// TIA Portal V17 export
// export: Created 2023-04-26T11:43:36.2466218Z, ExportSetting None, DisplayName Totally Integrated Automation Portal, DisplayVersion V17 Update 4, DisplayName TIA Portal Openness, DisplayVersion V17 Update 4, DisplayName TIA Portal Version Control Interface, DisplayVersion V17, DisplayName STEP 7 Professional, DisplayVersion V17 Update 4, DisplayName STEP 7 Safety, DisplayVersion V17, DisplayName WinCC Advanced / Unified PC, DisplayVersion V17 Update 4
FUNCTION "FC_AIn" : Void   // FC14, LAD
TITLE = FC_AIn
{ S7_Optimized_Access := 'FALSE' }
// Analog Input
// stored: SetENOAutomatically false
BEGIN

REGION Network 1: COMPRESSOR SUCTION PRESSURE
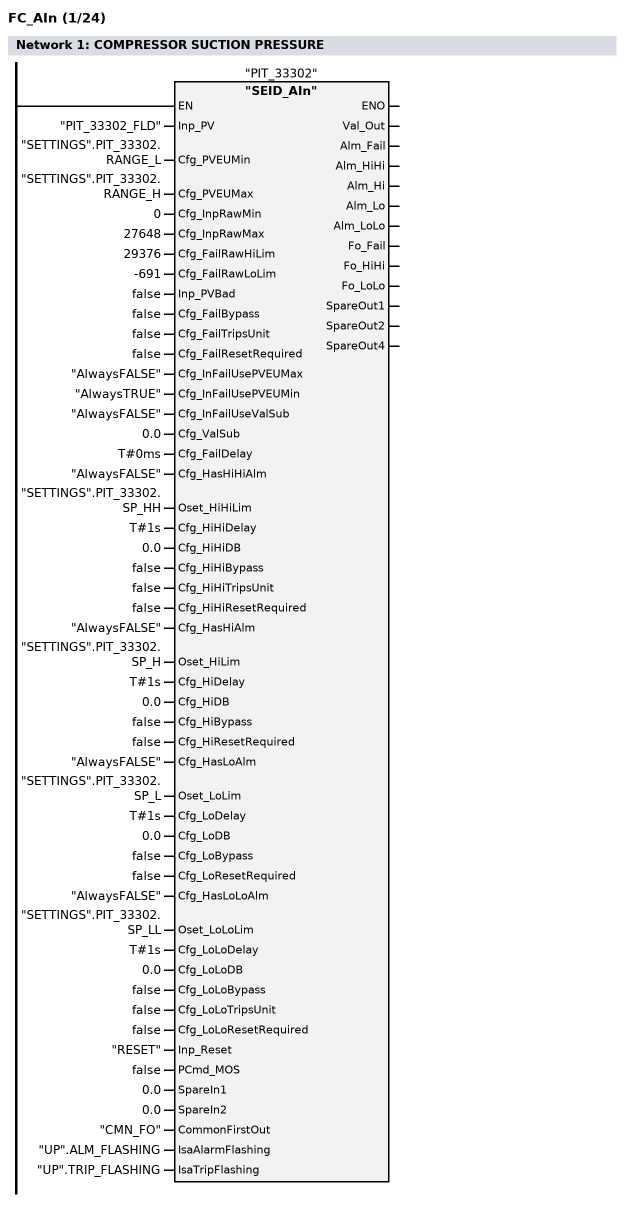
   RUNG wire#powerrail
      "PIT_33302"(Inp_PV := "PIT_33302_FLD", Cfg_PVEUMin := "SETTINGS".PIT_33302.RANGE_L, Cfg_PVEUMax := "SETTINGS".PIT_33302.RANGE_H, Cfg_InpRawMin := 0, Cfg_InpRawMax := 27648, Cfg_FailRawHiLim := 29376, Cfg_FailRawLoLim := -691, Inp_PVBad := false, Cfg_FailBypass := false, Cfg_FailTripsUnit := false, Cfg_FailResetRequired := false, Cfg_InFailUsePVEUMax := "AlwaysFALSE", Cfg_InFailUsePVEUMin := "AlwaysTRUE", Cfg_InFailUseValSub := "AlwaysFALSE", Cfg_ValSub := 0.0, Cfg_FailDelay := T#0ms, Cfg_HasHiHiAlm := "AlwaysFALSE", Oset_HiHiLim := "SETTINGS".PIT_33302.SP_HH, Cfg_HiHiDelay := T#1s, Cfg_HiHiDB := 0.0, Cfg_HiHiBypass := false, Cfg_HiHiTripsUnit := false, Cfg_HiHiResetRequired := false, Cfg_HasHiAlm := "AlwaysFALSE", Oset_HiLim := "SETTINGS".PIT_33302.SP_H, Cfg_HiDelay := T#1s, Cfg_HiDB := 0.0, Cfg_HiBypass := false, Cfg_HiResetRequired := false, Cfg_HasLoAlm := "AlwaysFALSE", Oset_LoLim := "SETTINGS".PIT_33302.SP_L, Cfg_LoDelay := T#1s, Cfg_LoDB := 0.0, Cfg_LoBypass := false, Cfg_LoResetRequired := false, Cfg_HasLoLoAlm := "AlwaysFALSE", Oset_LoLoLim := "SETTINGS".PIT_33302.SP_LL, Cfg_LoLoDelay := T#1s, Cfg_LoLoDB := 0.0, Cfg_LoLoBypass := false, Cfg_LoLoTripsUnit := false, Cfg_LoLoResetRequired := false, Inp_Reset := "RESET", PCmd_MOS := false, SpareIn1 := 0.0, SpareIn2 := 0.0, CommonFirstOut := "CMN_FO", IsaAlarmFlashing := "UP".ALM_FLASHING, IsaTripFlashing := "UP".TRIP_FLASHING, Val_Out =>, Alm_Fail =>, Alm_HiHi =>, Alm_Hi =>, Alm_Lo =>, Alm_LoLo =>, Fo_Fail =>, Fo_HiHi =>, Fo_LoLo =>, SpareOut1 =>, SpareOut2 =>, SpareOut4 =>)
   END_RUNG
   // the same network as SCL:
   "PIT_33302"(Inp_PV := "PIT_33302_FLD",   // "SEID_AIn"
               Cfg_PVEUMin := "SETTINGS".PIT_33302.RANGE_L,
               Cfg_PVEUMax := "SETTINGS".PIT_33302.RANGE_H,
               Cfg_InpRawMin := 0,
               Cfg_InpRawMax := 27648,
               Cfg_FailRawHiLim := 29376,
               Cfg_FailRawLoLim := -691,
               Inp_PVBad := false,
               Cfg_FailBypass := false,
               Cfg_FailTripsUnit := false,
               Cfg_FailResetRequired := false,
               Cfg_InFailUsePVEUMax := "AlwaysFALSE",
               Cfg_InFailUsePVEUMin := "AlwaysTRUE",
               Cfg_InFailUseValSub := "AlwaysFALSE",
               Cfg_ValSub := 0.0,
               Cfg_FailDelay := T#0ms,
               Cfg_HasHiHiAlm := "AlwaysFALSE",
               Oset_HiHiLim := "SETTINGS".PIT_33302.SP_HH,
               Cfg_HiHiDelay := T#1s,
               Cfg_HiHiDB := 0.0,
               Cfg_HiHiBypass := false,
               Cfg_HiHiTripsUnit := false,
               Cfg_HiHiResetRequired := false,
               Cfg_HasHiAlm := "AlwaysFALSE",
               Oset_HiLim := "SETTINGS".PIT_33302.SP_H,
               Cfg_HiDelay := T#1s,
               Cfg_HiDB := 0.0,
               Cfg_HiBypass := false,
               Cfg_HiResetRequired := false,
               Cfg_HasLoAlm := "AlwaysFALSE",
               Oset_LoLim := "SETTINGS".PIT_33302.SP_L,
               Cfg_LoDelay := T#1s,
               Cfg_LoDB := 0.0,
               Cfg_LoBypass := false,
               Cfg_LoResetRequired := false,
               Cfg_HasLoLoAlm := "AlwaysFALSE",
               Oset_LoLoLim := "SETTINGS".PIT_33302.SP_LL,
               Cfg_LoLoDelay := T#1s,
               Cfg_LoLoDB := 0.0,
               Cfg_LoLoBypass := false,
               Cfg_LoLoTripsUnit := false,
               Cfg_LoLoResetRequired := false,
               Inp_Reset := "RESET",
               PCmd_MOS := false,
               SpareIn1 := 0.0,
               SpareIn2 := 0.0,
               CommonFirstOut := "CMN_FO",
               IsaAlarmFlashing := "UP".ALM_FLASHING,
               IsaTripFlashing := "UP".TRIP_FLASHING);
END_REGION

REGION Network 2: LUBE OIL SEPARATOR OUTLET PRESSURE
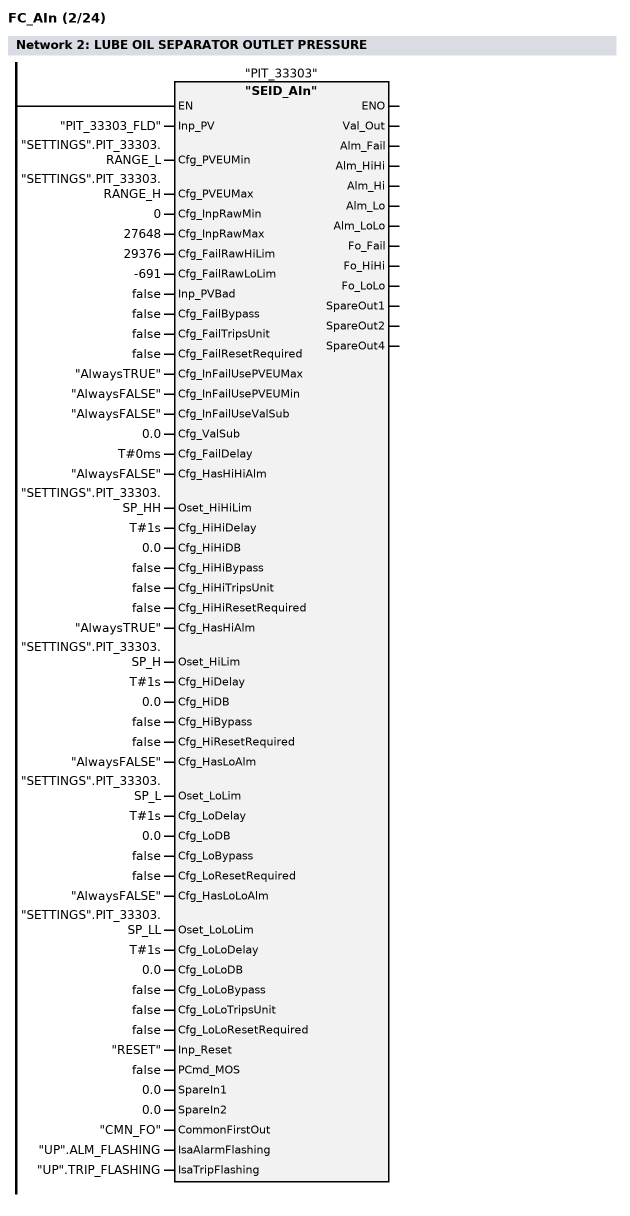
   RUNG wire#powerrail
      "PIT_33303"(Inp_PV := "PIT_33303_FLD", Cfg_PVEUMin := "SETTINGS".PIT_33303.RANGE_L, Cfg_PVEUMax := "SETTINGS".PIT_33303.RANGE_H, Cfg_InpRawMin := 0, Cfg_InpRawMax := 27648, Cfg_FailRawHiLim := 29376, Cfg_FailRawLoLim := -691, Inp_PVBad := false, Cfg_FailBypass := false, Cfg_FailTripsUnit := false, Cfg_FailResetRequired := false, Cfg_InFailUsePVEUMax := "AlwaysTRUE", Cfg_InFailUsePVEUMin := "AlwaysFALSE", Cfg_InFailUseValSub := "AlwaysFALSE", Cfg_ValSub := 0.0, Cfg_FailDelay := T#0ms, Cfg_HasHiHiAlm := "AlwaysFALSE", Oset_HiHiLim := "SETTINGS".PIT_33303.SP_HH, Cfg_HiHiDelay := T#1s, Cfg_HiHiDB := 0.0, Cfg_HiHiBypass := false, Cfg_HiHiTripsUnit := false, Cfg_HiHiResetRequired := false, Cfg_HasHiAlm := "AlwaysTRUE", Oset_HiLim := "SETTINGS".PIT_33303.SP_H, Cfg_HiDelay := T#1s, Cfg_HiDB := 0.0, Cfg_HiBypass := false, Cfg_HiResetRequired := false, Cfg_HasLoAlm := "AlwaysFALSE", Oset_LoLim := "SETTINGS".PIT_33303.SP_L, Cfg_LoDelay := T#1s, Cfg_LoDB := 0.0, Cfg_LoBypass := false, Cfg_LoResetRequired := false, Cfg_HasLoLoAlm := "AlwaysFALSE", Oset_LoLoLim := "SETTINGS".PIT_33303.SP_LL, Cfg_LoLoDelay := T#1s, Cfg_LoLoDB := 0.0, Cfg_LoLoBypass := false, Cfg_LoLoTripsUnit := false, Cfg_LoLoResetRequired := false, Inp_Reset := "RESET", PCmd_MOS := false, SpareIn1 := 0.0, SpareIn2 := 0.0, CommonFirstOut := "CMN_FO", IsaAlarmFlashing := "UP".ALM_FLASHING, IsaTripFlashing := "UP".TRIP_FLASHING, Val_Out =>, Alm_Fail =>, Alm_HiHi =>, Alm_Hi =>, Alm_Lo =>, Alm_LoLo =>, Fo_Fail =>, Fo_HiHi =>, Fo_LoLo =>, SpareOut1 =>, SpareOut2 =>, SpareOut4 =>)
   END_RUNG
   // the same network as SCL:
   "PIT_33303"(Inp_PV := "PIT_33303_FLD",   // "SEID_AIn"
               Cfg_PVEUMin := "SETTINGS".PIT_33303.RANGE_L,
               Cfg_PVEUMax := "SETTINGS".PIT_33303.RANGE_H,
               Cfg_InpRawMin := 0,
               Cfg_InpRawMax := 27648,
               Cfg_FailRawHiLim := 29376,
               Cfg_FailRawLoLim := -691,
               Inp_PVBad := false,
               Cfg_FailBypass := false,
               Cfg_FailTripsUnit := false,
               Cfg_FailResetRequired := false,
               Cfg_InFailUsePVEUMax := "AlwaysTRUE",
               Cfg_InFailUsePVEUMin := "AlwaysFALSE",
               Cfg_InFailUseValSub := "AlwaysFALSE",
               Cfg_ValSub := 0.0,
               Cfg_FailDelay := T#0ms,
               Cfg_HasHiHiAlm := "AlwaysFALSE",
               Oset_HiHiLim := "SETTINGS".PIT_33303.SP_HH,
               Cfg_HiHiDelay := T#1s,
               Cfg_HiHiDB := 0.0,
               Cfg_HiHiBypass := false,
               Cfg_HiHiTripsUnit := false,
               Cfg_HiHiResetRequired := false,
               Cfg_HasHiAlm := "AlwaysTRUE",
               Oset_HiLim := "SETTINGS".PIT_33303.SP_H,
               Cfg_HiDelay := T#1s,
               Cfg_HiDB := 0.0,
               Cfg_HiBypass := false,
               Cfg_HiResetRequired := false,
               Cfg_HasLoAlm := "AlwaysFALSE",
               Oset_LoLim := "SETTINGS".PIT_33303.SP_L,
               Cfg_LoDelay := T#1s,
               Cfg_LoDB := 0.0,
               Cfg_LoBypass := false,
               Cfg_LoResetRequired := false,
               Cfg_HasLoLoAlm := "AlwaysFALSE",
               Oset_LoLoLim := "SETTINGS".PIT_33303.SP_LL,
               Cfg_LoLoDelay := T#1s,
               Cfg_LoLoDB := 0.0,
               Cfg_LoLoBypass := false,
               Cfg_LoLoTripsUnit := false,
               Cfg_LoLoResetRequired := false,
               Inp_Reset := "RESET",
               PCmd_MOS := false,
               SpareIn1 := 0.0,
               SpareIn2 := 0.0,
               CommonFirstOut := "CMN_FO",
               IsaAlarmFlashing := "UP".ALM_FLASHING,
               IsaTripFlashing := "UP".TRIP_FLASHING);
END_REGION

REGION Network 3: CONDENSER LEVEL
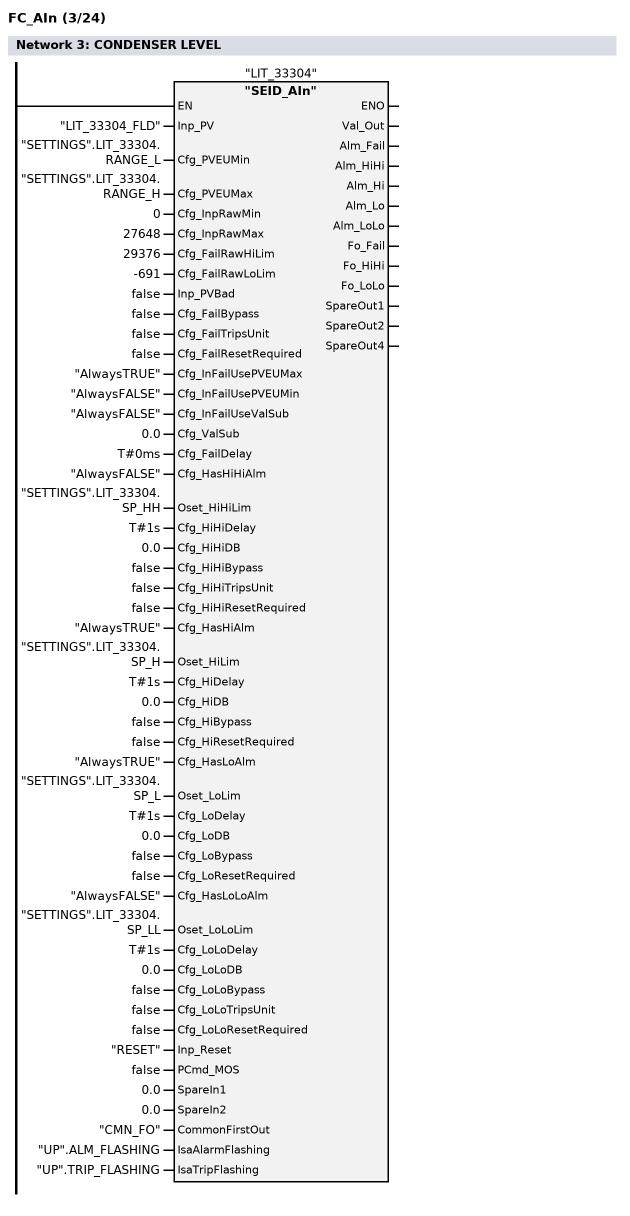
   RUNG wire#powerrail
      "LIT_33304"(Inp_PV := "LIT_33304_FLD", Cfg_PVEUMin := "SETTINGS".LIT_33304.RANGE_L, Cfg_PVEUMax := "SETTINGS".LIT_33304.RANGE_H, Cfg_InpRawMin := 0, Cfg_InpRawMax := 27648, Cfg_FailRawHiLim := 29376, Cfg_FailRawLoLim := -691, Inp_PVBad := false, Cfg_FailBypass := false, Cfg_FailTripsUnit := false, Cfg_FailResetRequired := false, Cfg_InFailUsePVEUMax := "AlwaysTRUE", Cfg_InFailUsePVEUMin := "AlwaysFALSE", Cfg_InFailUseValSub := "AlwaysFALSE", Cfg_ValSub := 0.0, Cfg_FailDelay := T#0ms, Cfg_HasHiHiAlm := "AlwaysFALSE", Oset_HiHiLim := "SETTINGS".LIT_33304.SP_HH, Cfg_HiHiDelay := T#1s, Cfg_HiHiDB := 0.0, Cfg_HiHiBypass := false, Cfg_HiHiTripsUnit := false, Cfg_HiHiResetRequired := false, Cfg_HasHiAlm := "AlwaysTRUE", Oset_HiLim := "SETTINGS".LIT_33304.SP_H, Cfg_HiDelay := T#1s, Cfg_HiDB := 0.0, Cfg_HiBypass := false, Cfg_HiResetRequired := false, Cfg_HasLoAlm := "AlwaysTRUE", Oset_LoLim := "SETTINGS".LIT_33304.SP_L, Cfg_LoDelay := T#1s, Cfg_LoDB := 0.0, Cfg_LoBypass := false, Cfg_LoResetRequired := false, Cfg_HasLoLoAlm := "AlwaysFALSE", Oset_LoLoLim := "SETTINGS".LIT_33304.SP_LL, Cfg_LoLoDelay := T#1s, Cfg_LoLoDB := 0.0, Cfg_LoLoBypass := false, Cfg_LoLoTripsUnit := false, Cfg_LoLoResetRequired := false, Inp_Reset := "RESET", PCmd_MOS := false, SpareIn1 := 0.0, SpareIn2 := 0.0, CommonFirstOut := "CMN_FO", IsaAlarmFlashing := "UP".ALM_FLASHING, IsaTripFlashing := "UP".TRIP_FLASHING, Val_Out =>, Alm_Fail =>, Alm_HiHi =>, Alm_Hi =>, Alm_Lo =>, Alm_LoLo =>, Fo_Fail =>, Fo_HiHi =>, Fo_LoLo =>, SpareOut1 =>, SpareOut2 =>, SpareOut4 =>)
   END_RUNG
   // the same network as SCL:
   "LIT_33304"(Inp_PV := "LIT_33304_FLD",   // "SEID_AIn"
               Cfg_PVEUMin := "SETTINGS".LIT_33304.RANGE_L,
               Cfg_PVEUMax := "SETTINGS".LIT_33304.RANGE_H,
               Cfg_InpRawMin := 0,
               Cfg_InpRawMax := 27648,
               Cfg_FailRawHiLim := 29376,
               Cfg_FailRawLoLim := -691,
               Inp_PVBad := false,
               Cfg_FailBypass := false,
               Cfg_FailTripsUnit := false,
               Cfg_FailResetRequired := false,
               Cfg_InFailUsePVEUMax := "AlwaysTRUE",
               Cfg_InFailUsePVEUMin := "AlwaysFALSE",
               Cfg_InFailUseValSub := "AlwaysFALSE",
               Cfg_ValSub := 0.0,
               Cfg_FailDelay := T#0ms,
               Cfg_HasHiHiAlm := "AlwaysFALSE",
               Oset_HiHiLim := "SETTINGS".LIT_33304.SP_HH,
               Cfg_HiHiDelay := T#1s,
               Cfg_HiHiDB := 0.0,
               Cfg_HiHiBypass := false,
               Cfg_HiHiTripsUnit := false,
               Cfg_HiHiResetRequired := false,
               Cfg_HasHiAlm := "AlwaysTRUE",
               Oset_HiLim := "SETTINGS".LIT_33304.SP_H,
               Cfg_HiDelay := T#1s,
               Cfg_HiDB := 0.0,
               Cfg_HiBypass := false,
               Cfg_HiResetRequired := false,
               Cfg_HasLoAlm := "AlwaysTRUE",
               Oset_LoLim := "SETTINGS".LIT_33304.SP_L,
               Cfg_LoDelay := T#1s,
               Cfg_LoDB := 0.0,
               Cfg_LoBypass := false,
               Cfg_LoResetRequired := false,
               Cfg_HasLoLoAlm := "AlwaysFALSE",
               Oset_LoLoLim := "SETTINGS".LIT_33304.SP_LL,
               Cfg_LoLoDelay := T#1s,
               Cfg_LoLoDB := 0.0,
               Cfg_LoLoBypass := false,
               Cfg_LoLoTripsUnit := false,
               Cfg_LoLoResetRequired := false,
               Inp_Reset := "RESET",
               PCmd_MOS := false,
               SpareIn1 := 0.0,
               SpareIn2 := 0.0,
               CommonFirstOut := "CMN_FO",
               IsaAlarmFlashing := "UP".ALM_FLASHING,
               IsaTripFlashing := "UP".TRIP_FLASHING);
END_REGION

REGION Network 4: COMPRESSOR SUCTION PRESSURE
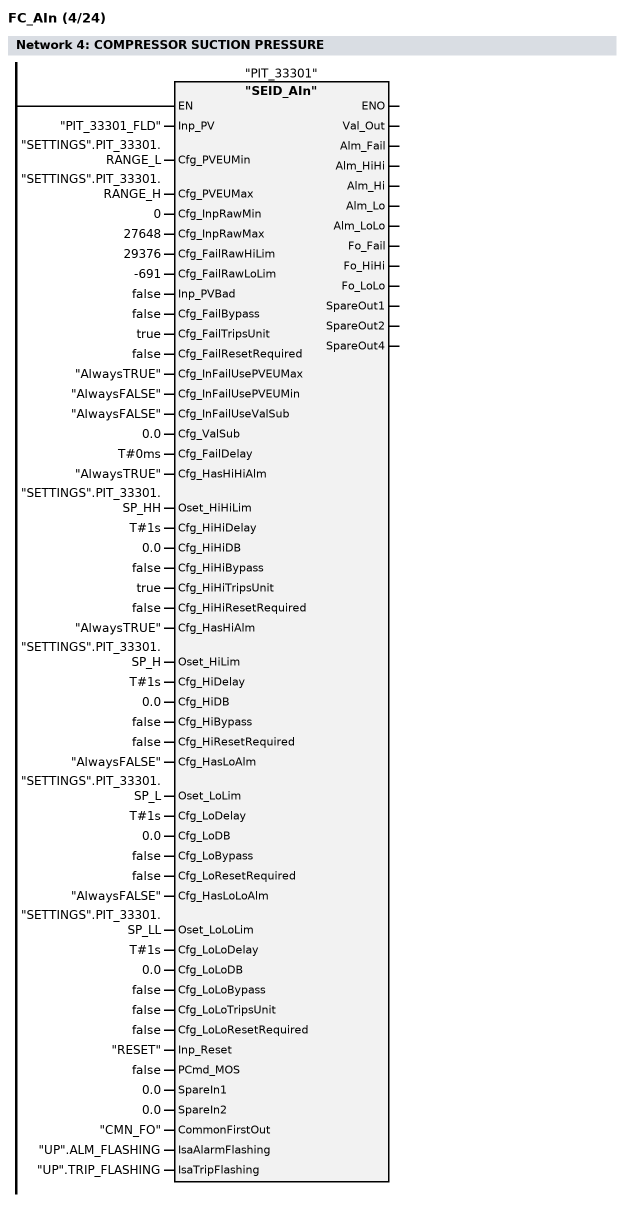
   RUNG wire#powerrail
      "PIT_33301"(Inp_PV := "PIT_33301_FLD", Cfg_PVEUMin := "SETTINGS".PIT_33301.RANGE_L, Cfg_PVEUMax := "SETTINGS".PIT_33301.RANGE_H, Cfg_InpRawMin := 0, Cfg_InpRawMax := 27648, Cfg_FailRawHiLim := 29376, Cfg_FailRawLoLim := -691, Inp_PVBad := false, Cfg_FailBypass := false, Cfg_FailTripsUnit := true, Cfg_FailResetRequired := false, Cfg_InFailUsePVEUMax := "AlwaysTRUE", Cfg_InFailUsePVEUMin := "AlwaysFALSE", Cfg_InFailUseValSub := "AlwaysFALSE", Cfg_ValSub := 0.0, Cfg_FailDelay := T#0ms, Cfg_HasHiHiAlm := "AlwaysTRUE", Oset_HiHiLim := "SETTINGS".PIT_33301.SP_HH, Cfg_HiHiDelay := T#1s, Cfg_HiHiDB := 0.0, Cfg_HiHiBypass := false, Cfg_HiHiTripsUnit := true, Cfg_HiHiResetRequired := false, Cfg_HasHiAlm := "AlwaysTRUE", Oset_HiLim := "SETTINGS".PIT_33301.SP_H, Cfg_HiDelay := T#1s, Cfg_HiDB := 0.0, Cfg_HiBypass := false, Cfg_HiResetRequired := false, Cfg_HasLoAlm := "AlwaysFALSE", Oset_LoLim := "SETTINGS".PIT_33301.SP_L, Cfg_LoDelay := T#1s, Cfg_LoDB := 0.0, Cfg_LoBypass := false, Cfg_LoResetRequired := false, Cfg_HasLoLoAlm := "AlwaysFALSE", Oset_LoLoLim := "SETTINGS".PIT_33301.SP_LL, Cfg_LoLoDelay := T#1s, Cfg_LoLoDB := 0.0, Cfg_LoLoBypass := false, Cfg_LoLoTripsUnit := false, Cfg_LoLoResetRequired := false, Inp_Reset := "RESET", PCmd_MOS := false, SpareIn1 := 0.0, SpareIn2 := 0.0, CommonFirstOut := "CMN_FO", IsaAlarmFlashing := "UP".ALM_FLASHING, IsaTripFlashing := "UP".TRIP_FLASHING, Val_Out =>, Alm_Fail =>, Alm_HiHi =>, Alm_Hi =>, Alm_Lo =>, Alm_LoLo =>, Fo_Fail =>, Fo_HiHi =>, Fo_LoLo =>, SpareOut1 =>, SpareOut2 =>, SpareOut4 =>)
   END_RUNG
   // the same network as SCL:
   "PIT_33301"(Inp_PV := "PIT_33301_FLD",   // "SEID_AIn"
               Cfg_PVEUMin := "SETTINGS".PIT_33301.RANGE_L,
               Cfg_PVEUMax := "SETTINGS".PIT_33301.RANGE_H,
               Cfg_InpRawMin := 0,
               Cfg_InpRawMax := 27648,
               Cfg_FailRawHiLim := 29376,
               Cfg_FailRawLoLim := -691,
               Inp_PVBad := false,
               Cfg_FailBypass := false,
               Cfg_FailTripsUnit := true,
               Cfg_FailResetRequired := false,
               Cfg_InFailUsePVEUMax := "AlwaysTRUE",
               Cfg_InFailUsePVEUMin := "AlwaysFALSE",
               Cfg_InFailUseValSub := "AlwaysFALSE",
               Cfg_ValSub := 0.0,
               Cfg_FailDelay := T#0ms,
               Cfg_HasHiHiAlm := "AlwaysTRUE",
               Oset_HiHiLim := "SETTINGS".PIT_33301.SP_HH,
               Cfg_HiHiDelay := T#1s,
               Cfg_HiHiDB := 0.0,
               Cfg_HiHiBypass := false,
               Cfg_HiHiTripsUnit := true,
               Cfg_HiHiResetRequired := false,
               Cfg_HasHiAlm := "AlwaysTRUE",
               Oset_HiLim := "SETTINGS".PIT_33301.SP_H,
               Cfg_HiDelay := T#1s,
               Cfg_HiDB := 0.0,
               Cfg_HiBypass := false,
               Cfg_HiResetRequired := false,
               Cfg_HasLoAlm := "AlwaysFALSE",
               Oset_LoLim := "SETTINGS".PIT_33301.SP_L,
               Cfg_LoDelay := T#1s,
               Cfg_LoDB := 0.0,
               Cfg_LoBypass := false,
               Cfg_LoResetRequired := false,
               Cfg_HasLoLoAlm := "AlwaysFALSE",
               Oset_LoLoLim := "SETTINGS".PIT_33301.SP_LL,
               Cfg_LoLoDelay := T#1s,
               Cfg_LoLoDB := 0.0,
               Cfg_LoLoBypass := false,
               Cfg_LoLoTripsUnit := false,
               Cfg_LoLoResetRequired := false,
               Inp_Reset := "RESET",
               PCmd_MOS := false,
               SpareIn1 := 0.0,
               SpareIn2 := 0.0,
               CommonFirstOut := "CMN_FO",
               IsaAlarmFlashing := "UP".ALM_FLASHING,
               IsaTripFlashing := "UP".TRIP_FLASHING);
END_REGION

REGION Network 5: LUBE OIL SEPARATOR OUTLET TEMPERATURE
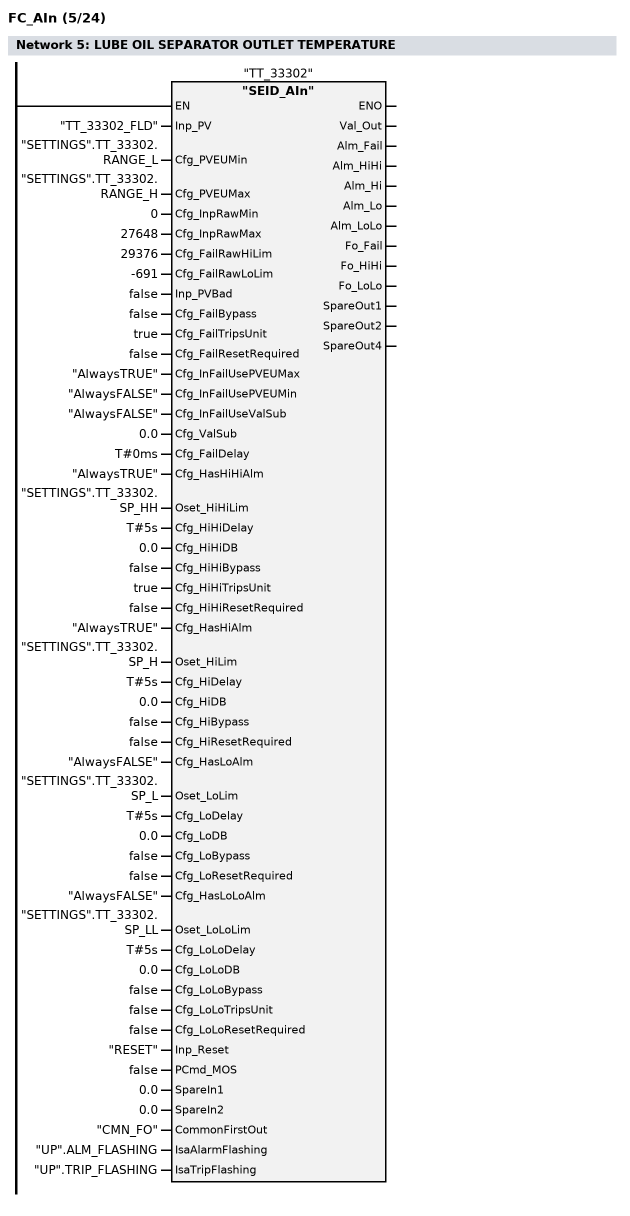
   RUNG wire#powerrail
      "TT_33302"(Inp_PV := "TT_33302_FLD", Cfg_PVEUMin := "SETTINGS".TT_33302.RANGE_L, Cfg_PVEUMax := "SETTINGS".TT_33302.RANGE_H, Cfg_InpRawMin := 0, Cfg_InpRawMax := 27648, Cfg_FailRawHiLim := 29376, Cfg_FailRawLoLim := -691, Inp_PVBad := false, Cfg_FailBypass := false, Cfg_FailTripsUnit := true, Cfg_FailResetRequired := false, Cfg_InFailUsePVEUMax := "AlwaysTRUE", Cfg_InFailUsePVEUMin := "AlwaysFALSE", Cfg_InFailUseValSub := "AlwaysFALSE", Cfg_ValSub := 0.0, Cfg_FailDelay := T#0ms, Cfg_HasHiHiAlm := "AlwaysTRUE", Oset_HiHiLim := "SETTINGS".TT_33302.SP_HH, Cfg_HiHiDelay := T#5s, Cfg_HiHiDB := 0.0, Cfg_HiHiBypass := false, Cfg_HiHiTripsUnit := true, Cfg_HiHiResetRequired := false, Cfg_HasHiAlm := "AlwaysTRUE", Oset_HiLim := "SETTINGS".TT_33302.SP_H, Cfg_HiDelay := T#5s, Cfg_HiDB := 0.0, Cfg_HiBypass := false, Cfg_HiResetRequired := false, Cfg_HasLoAlm := "AlwaysFALSE", Oset_LoLim := "SETTINGS".TT_33302.SP_L, Cfg_LoDelay := T#5s, Cfg_LoDB := 0.0, Cfg_LoBypass := false, Cfg_LoResetRequired := false, Cfg_HasLoLoAlm := "AlwaysFALSE", Oset_LoLoLim := "SETTINGS".TT_33302.SP_LL, Cfg_LoLoDelay := T#5s, Cfg_LoLoDB := 0.0, Cfg_LoLoBypass := false, Cfg_LoLoTripsUnit := false, Cfg_LoLoResetRequired := false, Inp_Reset := "RESET", PCmd_MOS := false, SpareIn1 := 0.0, SpareIn2 := 0.0, CommonFirstOut := "CMN_FO", IsaAlarmFlashing := "UP".ALM_FLASHING, IsaTripFlashing := "UP".TRIP_FLASHING, Val_Out =>, Alm_Fail =>, Alm_HiHi =>, Alm_Hi =>, Alm_Lo =>, Alm_LoLo =>, Fo_Fail =>, Fo_HiHi =>, Fo_LoLo =>, SpareOut1 =>, SpareOut2 =>, SpareOut4 =>)
   END_RUNG
   // the same network as SCL:
   "TT_33302"(Inp_PV := "TT_33302_FLD",   // "SEID_AIn"
              Cfg_PVEUMin := "SETTINGS".TT_33302.RANGE_L,
              Cfg_PVEUMax := "SETTINGS".TT_33302.RANGE_H,
              Cfg_InpRawMin := 0,
              Cfg_InpRawMax := 27648,
              Cfg_FailRawHiLim := 29376,
              Cfg_FailRawLoLim := -691,
              Inp_PVBad := false,
              Cfg_FailBypass := false,
              Cfg_FailTripsUnit := true,
              Cfg_FailResetRequired := false,
              Cfg_InFailUsePVEUMax := "AlwaysTRUE",
              Cfg_InFailUsePVEUMin := "AlwaysFALSE",
              Cfg_InFailUseValSub := "AlwaysFALSE",
              Cfg_ValSub := 0.0,
              Cfg_FailDelay := T#0ms,
              Cfg_HasHiHiAlm := "AlwaysTRUE",
              Oset_HiHiLim := "SETTINGS".TT_33302.SP_HH,
              Cfg_HiHiDelay := T#5s,
              Cfg_HiHiDB := 0.0,
              Cfg_HiHiBypass := false,
              Cfg_HiHiTripsUnit := true,
              Cfg_HiHiResetRequired := false,
              Cfg_HasHiAlm := "AlwaysTRUE",
              Oset_HiLim := "SETTINGS".TT_33302.SP_H,
              Cfg_HiDelay := T#5s,
              Cfg_HiDB := 0.0,
              Cfg_HiBypass := false,
              Cfg_HiResetRequired := false,
              Cfg_HasLoAlm := "AlwaysFALSE",
              Oset_LoLim := "SETTINGS".TT_33302.SP_L,
              Cfg_LoDelay := T#5s,
              Cfg_LoDB := 0.0,
              Cfg_LoBypass := false,
              Cfg_LoResetRequired := false,
              Cfg_HasLoLoAlm := "AlwaysFALSE",
              Oset_LoLoLim := "SETTINGS".TT_33302.SP_LL,
              Cfg_LoLoDelay := T#5s,
              Cfg_LoLoDB := 0.0,
              Cfg_LoLoBypass := false,
              Cfg_LoLoTripsUnit := false,
              Cfg_LoLoResetRequired := false,
              Inp_Reset := "RESET",
              PCmd_MOS := false,
              SpareIn1 := 0.0,
              SpareIn2 := 0.0,
              CommonFirstOut := "CMN_FO",
              IsaAlarmFlashing := "UP".ALM_FLASHING,
              IsaTripFlashing := "UP".TRIP_FLASHING);
END_REGION

REGION Network 6: LUBE OIL SEPARATOR OUTLET PRESSURE
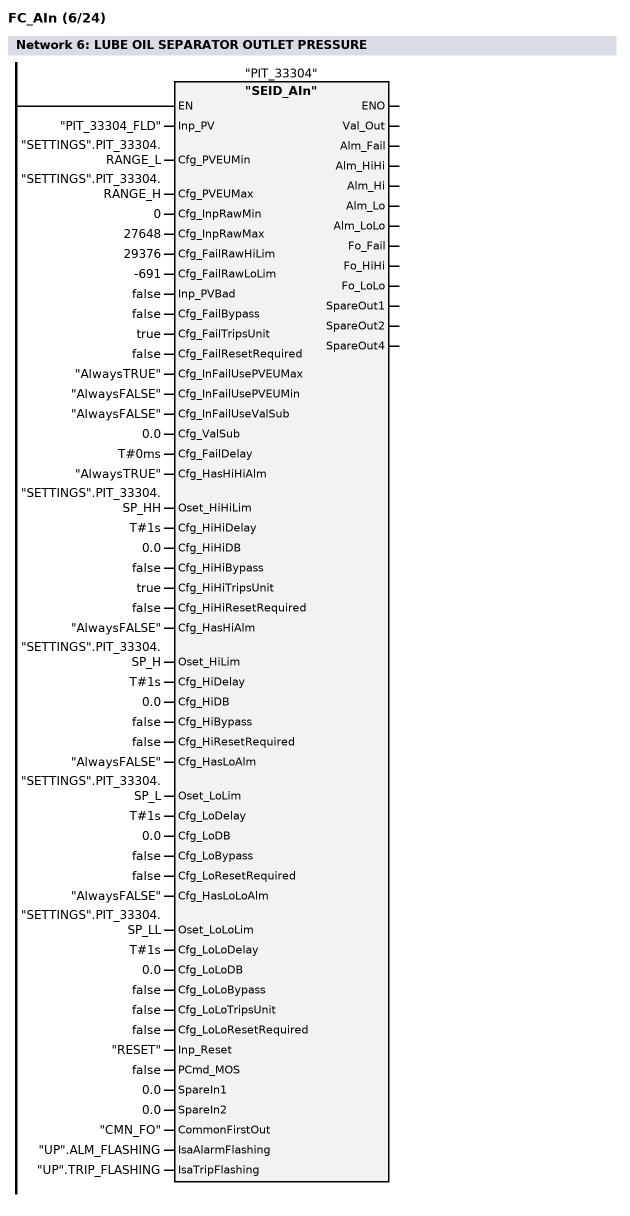
   RUNG wire#powerrail
      "PIT_33304"(Inp_PV := "PIT_33304_FLD", Cfg_PVEUMin := "SETTINGS".PIT_33304.RANGE_L, Cfg_PVEUMax := "SETTINGS".PIT_33304.RANGE_H, Cfg_InpRawMin := 0, Cfg_InpRawMax := 27648, Cfg_FailRawHiLim := 29376, Cfg_FailRawLoLim := -691, Inp_PVBad := false, Cfg_FailBypass := false, Cfg_FailTripsUnit := true, Cfg_FailResetRequired := false, Cfg_InFailUsePVEUMax := "AlwaysTRUE", Cfg_InFailUsePVEUMin := "AlwaysFALSE", Cfg_InFailUseValSub := "AlwaysFALSE", Cfg_ValSub := 0.0, Cfg_FailDelay := T#0ms, Cfg_HasHiHiAlm := "AlwaysTRUE", Oset_HiHiLim := "SETTINGS".PIT_33304.SP_HH, Cfg_HiHiDelay := T#1s, Cfg_HiHiDB := 0.0, Cfg_HiHiBypass := false, Cfg_HiHiTripsUnit := true, Cfg_HiHiResetRequired := false, Cfg_HasHiAlm := "AlwaysFALSE", Oset_HiLim := "SETTINGS".PIT_33304.SP_H, Cfg_HiDelay := T#1s, Cfg_HiDB := 0.0, Cfg_HiBypass := false, Cfg_HiResetRequired := false, Cfg_HasLoAlm := "AlwaysFALSE", Oset_LoLim := "SETTINGS".PIT_33304.SP_L, Cfg_LoDelay := T#1s, Cfg_LoDB := 0.0, Cfg_LoBypass := false, Cfg_LoResetRequired := false, Cfg_HasLoLoAlm := "AlwaysFALSE", Oset_LoLoLim := "SETTINGS".PIT_33304.SP_LL, Cfg_LoLoDelay := T#1s, Cfg_LoLoDB := 0.0, Cfg_LoLoBypass := false, Cfg_LoLoTripsUnit := false, Cfg_LoLoResetRequired := false, Inp_Reset := "RESET", PCmd_MOS := false, SpareIn1 := 0.0, SpareIn2 := 0.0, CommonFirstOut := "CMN_FO", IsaAlarmFlashing := "UP".ALM_FLASHING, IsaTripFlashing := "UP".TRIP_FLASHING, Val_Out =>, Alm_Fail =>, Alm_HiHi =>, Alm_Hi =>, Alm_Lo =>, Alm_LoLo =>, Fo_Fail =>, Fo_HiHi =>, Fo_LoLo =>, SpareOut1 =>, SpareOut2 =>, SpareOut4 =>)
   END_RUNG
   // the same network as SCL:
   "PIT_33304"(Inp_PV := "PIT_33304_FLD",   // "SEID_AIn"
               Cfg_PVEUMin := "SETTINGS".PIT_33304.RANGE_L,
               Cfg_PVEUMax := "SETTINGS".PIT_33304.RANGE_H,
               Cfg_InpRawMin := 0,
               Cfg_InpRawMax := 27648,
               Cfg_FailRawHiLim := 29376,
               Cfg_FailRawLoLim := -691,
               Inp_PVBad := false,
               Cfg_FailBypass := false,
               Cfg_FailTripsUnit := true,
               Cfg_FailResetRequired := false,
               Cfg_InFailUsePVEUMax := "AlwaysTRUE",
               Cfg_InFailUsePVEUMin := "AlwaysFALSE",
               Cfg_InFailUseValSub := "AlwaysFALSE",
               Cfg_ValSub := 0.0,
               Cfg_FailDelay := T#0ms,
               Cfg_HasHiHiAlm := "AlwaysTRUE",
               Oset_HiHiLim := "SETTINGS".PIT_33304.SP_HH,
               Cfg_HiHiDelay := T#1s,
               Cfg_HiHiDB := 0.0,
               Cfg_HiHiBypass := false,
               Cfg_HiHiTripsUnit := true,
               Cfg_HiHiResetRequired := false,
               Cfg_HasHiAlm := "AlwaysFALSE",
               Oset_HiLim := "SETTINGS".PIT_33304.SP_H,
               Cfg_HiDelay := T#1s,
               Cfg_HiDB := 0.0,
               Cfg_HiBypass := false,
               Cfg_HiResetRequired := false,
               Cfg_HasLoAlm := "AlwaysFALSE",
               Oset_LoLim := "SETTINGS".PIT_33304.SP_L,
               Cfg_LoDelay := T#1s,
               Cfg_LoDB := 0.0,
               Cfg_LoBypass := false,
               Cfg_LoResetRequired := false,
               Cfg_HasLoLoAlm := "AlwaysFALSE",
               Oset_LoLoLim := "SETTINGS".PIT_33304.SP_LL,
               Cfg_LoLoDelay := T#1s,
               Cfg_LoLoDB := 0.0,
               Cfg_LoLoBypass := false,
               Cfg_LoLoTripsUnit := false,
               Cfg_LoLoResetRequired := false,
               Inp_Reset := "RESET",
               PCmd_MOS := false,
               SpareIn1 := 0.0,
               SpareIn2 := 0.0,
               CommonFirstOut := "CMN_FO",
               IsaAlarmFlashing := "UP".ALM_FLASHING,
               IsaTripFlashing := "UP".TRIP_FLASHING);
END_REGION

REGION Network 7: OIL DIFFERENTIAL PRESSURE
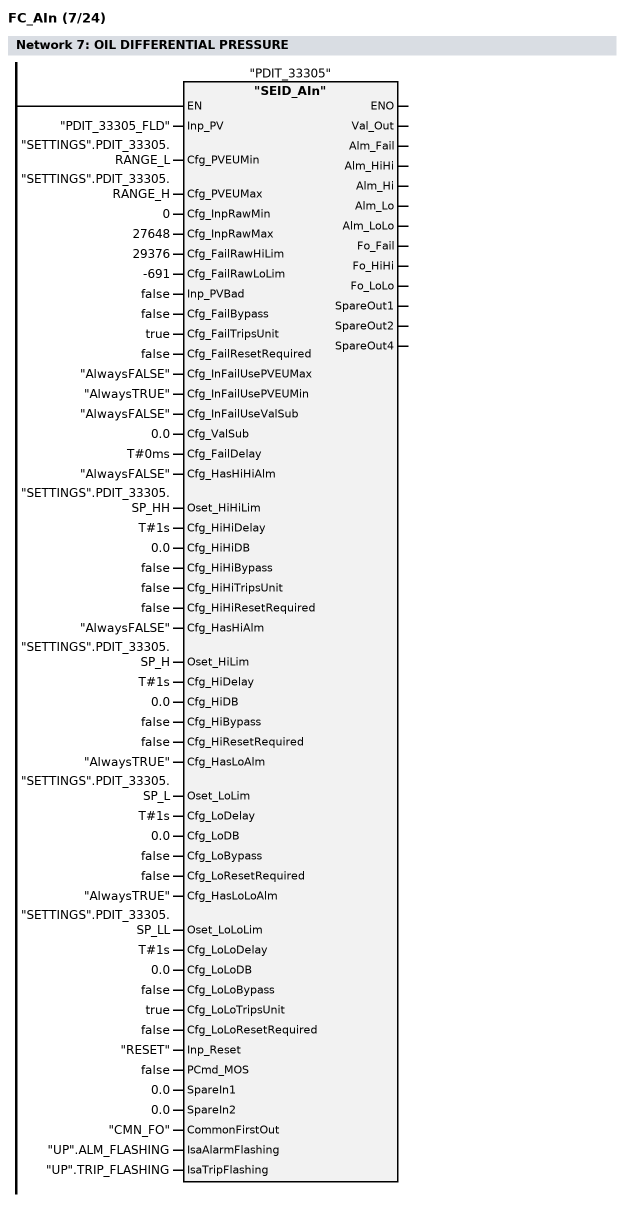
   RUNG wire#powerrail
      "PDIT_33305"(Inp_PV := "PDIT_33305_FLD", Cfg_PVEUMin := "SETTINGS".PDIT_33305.RANGE_L, Cfg_PVEUMax := "SETTINGS".PDIT_33305.RANGE_H, Cfg_InpRawMin := 0, Cfg_InpRawMax := 27648, Cfg_FailRawHiLim := 29376, Cfg_FailRawLoLim := -691, Inp_PVBad := false, Cfg_FailBypass := false, Cfg_FailTripsUnit := true, Cfg_FailResetRequired := false, Cfg_InFailUsePVEUMax := "AlwaysFALSE", Cfg_InFailUsePVEUMin := "AlwaysTRUE", Cfg_InFailUseValSub := "AlwaysFALSE", Cfg_ValSub := 0.0, Cfg_FailDelay := T#0ms, Cfg_HasHiHiAlm := "AlwaysFALSE", Oset_HiHiLim := "SETTINGS".PDIT_33305.SP_HH, Cfg_HiHiDelay := T#1s, Cfg_HiHiDB := 0.0, Cfg_HiHiBypass := false, Cfg_HiHiTripsUnit := false, Cfg_HiHiResetRequired := false, Cfg_HasHiAlm := "AlwaysFALSE", Oset_HiLim := "SETTINGS".PDIT_33305.SP_H, Cfg_HiDelay := T#1s, Cfg_HiDB := 0.0, Cfg_HiBypass := false, Cfg_HiResetRequired := false, Cfg_HasLoAlm := "AlwaysTRUE", Oset_LoLim := "SETTINGS".PDIT_33305.SP_L, Cfg_LoDelay := T#1s, Cfg_LoDB := 0.0, Cfg_LoBypass := false, Cfg_LoResetRequired := false, Cfg_HasLoLoAlm := "AlwaysTRUE", Oset_LoLoLim := "SETTINGS".PDIT_33305.SP_LL, Cfg_LoLoDelay := T#1s, Cfg_LoLoDB := 0.0, Cfg_LoLoBypass := false, Cfg_LoLoTripsUnit := true, Cfg_LoLoResetRequired := false, Inp_Reset := "RESET", PCmd_MOS := false, SpareIn1 := 0.0, SpareIn2 := 0.0, CommonFirstOut := "CMN_FO", IsaAlarmFlashing := "UP".ALM_FLASHING, IsaTripFlashing := "UP".TRIP_FLASHING, Val_Out =>, Alm_Fail =>, Alm_HiHi =>, Alm_Hi =>, Alm_Lo =>, Alm_LoLo =>, Fo_Fail =>, Fo_HiHi =>, Fo_LoLo =>, SpareOut1 =>, SpareOut2 =>, SpareOut4 =>)
   END_RUNG
   // the same network as SCL:
   "PDIT_33305"(Inp_PV := "PDIT_33305_FLD",   // "SEID_AIn"
                Cfg_PVEUMin := "SETTINGS".PDIT_33305.RANGE_L,
                Cfg_PVEUMax := "SETTINGS".PDIT_33305.RANGE_H,
                Cfg_InpRawMin := 0,
                Cfg_InpRawMax := 27648,
                Cfg_FailRawHiLim := 29376,
                Cfg_FailRawLoLim := -691,
                Inp_PVBad := false,
                Cfg_FailBypass := false,
                Cfg_FailTripsUnit := true,
                Cfg_FailResetRequired := false,
                Cfg_InFailUsePVEUMax := "AlwaysFALSE",
                Cfg_InFailUsePVEUMin := "AlwaysTRUE",
                Cfg_InFailUseValSub := "AlwaysFALSE",
                Cfg_ValSub := 0.0,
                Cfg_FailDelay := T#0ms,
                Cfg_HasHiHiAlm := "AlwaysFALSE",
                Oset_HiHiLim := "SETTINGS".PDIT_33305.SP_HH,
                Cfg_HiHiDelay := T#1s,
                Cfg_HiHiDB := 0.0,
                Cfg_HiHiBypass := false,
                Cfg_HiHiTripsUnit := false,
                Cfg_HiHiResetRequired := false,
                Cfg_HasHiAlm := "AlwaysFALSE",
                Oset_HiLim := "SETTINGS".PDIT_33305.SP_H,
                Cfg_HiDelay := T#1s,
                Cfg_HiDB := 0.0,
                Cfg_HiBypass := false,
                Cfg_HiResetRequired := false,
                Cfg_HasLoAlm := "AlwaysTRUE",
                Oset_LoLim := "SETTINGS".PDIT_33305.SP_L,
                Cfg_LoDelay := T#1s,
                Cfg_LoDB := 0.0,
                Cfg_LoBypass := false,
                Cfg_LoResetRequired := false,
                Cfg_HasLoLoAlm := "AlwaysTRUE",
                Oset_LoLoLim := "SETTINGS".PDIT_33305.SP_LL,
                Cfg_LoLoDelay := T#1s,
                Cfg_LoLoDB := 0.0,
                Cfg_LoLoBypass := false,
                Cfg_LoLoTripsUnit := true,
                Cfg_LoLoResetRequired := false,
                Inp_Reset := "RESET",
                PCmd_MOS := false,
                SpareIn1 := 0.0,
                SpareIn2 := 0.0,
                CommonFirstOut := "CMN_FO",
                IsaAlarmFlashing := "UP".ALM_FLASHING,
                IsaTripFlashing := "UP".TRIP_FLASHING);
END_REGION

REGION Network 8: OIL TEMPERATURE
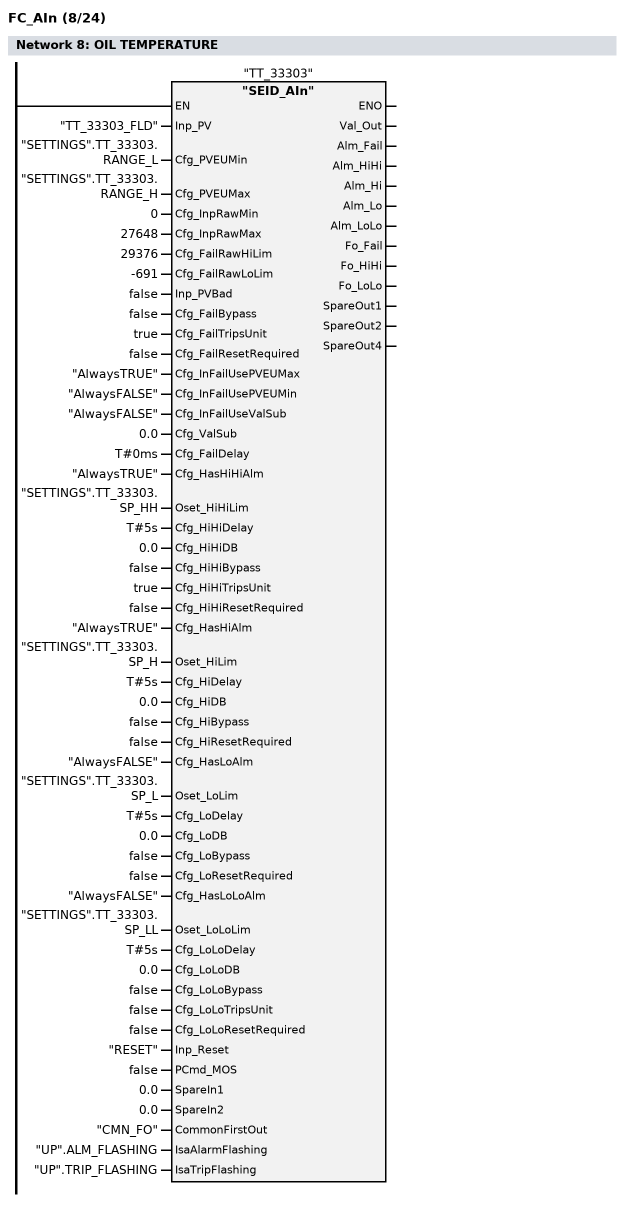
   RUNG wire#powerrail
      "TT_33303"(Inp_PV := "TT_33303_FLD", Cfg_PVEUMin := "SETTINGS".TT_33303.RANGE_L, Cfg_PVEUMax := "SETTINGS".TT_33303.RANGE_H, Cfg_InpRawMin := 0, Cfg_InpRawMax := 27648, Cfg_FailRawHiLim := 29376, Cfg_FailRawLoLim := -691, Inp_PVBad := false, Cfg_FailBypass := false, Cfg_FailTripsUnit := true, Cfg_FailResetRequired := false, Cfg_InFailUsePVEUMax := "AlwaysTRUE", Cfg_InFailUsePVEUMin := "AlwaysFALSE", Cfg_InFailUseValSub := "AlwaysFALSE", Cfg_ValSub := 0.0, Cfg_FailDelay := T#0ms, Cfg_HasHiHiAlm := "AlwaysTRUE", Oset_HiHiLim := "SETTINGS".TT_33303.SP_HH, Cfg_HiHiDelay := T#5s, Cfg_HiHiDB := 0.0, Cfg_HiHiBypass := false, Cfg_HiHiTripsUnit := true, Cfg_HiHiResetRequired := false, Cfg_HasHiAlm := "AlwaysTRUE", Oset_HiLim := "SETTINGS".TT_33303.SP_H, Cfg_HiDelay := T#5s, Cfg_HiDB := 0.0, Cfg_HiBypass := false, Cfg_HiResetRequired := false, Cfg_HasLoAlm := "AlwaysFALSE", Oset_LoLim := "SETTINGS".TT_33303.SP_L, Cfg_LoDelay := T#5s, Cfg_LoDB := 0.0, Cfg_LoBypass := false, Cfg_LoResetRequired := false, Cfg_HasLoLoAlm := "AlwaysFALSE", Oset_LoLoLim := "SETTINGS".TT_33303.SP_LL, Cfg_LoLoDelay := T#5s, Cfg_LoLoDB := 0.0, Cfg_LoLoBypass := false, Cfg_LoLoTripsUnit := false, Cfg_LoLoResetRequired := false, Inp_Reset := "RESET", PCmd_MOS := false, SpareIn1 := 0.0, SpareIn2 := 0.0, CommonFirstOut := "CMN_FO", IsaAlarmFlashing := "UP".ALM_FLASHING, IsaTripFlashing := "UP".TRIP_FLASHING, Val_Out =>, Alm_Fail =>, Alm_HiHi =>, Alm_Hi =>, Alm_Lo =>, Alm_LoLo =>, Fo_Fail =>, Fo_HiHi =>, Fo_LoLo =>, SpareOut1 =>, SpareOut2 =>, SpareOut4 =>)
   END_RUNG
   // the same network as SCL:
   "TT_33303"(Inp_PV := "TT_33303_FLD",   // "SEID_AIn"
              Cfg_PVEUMin := "SETTINGS".TT_33303.RANGE_L,
              Cfg_PVEUMax := "SETTINGS".TT_33303.RANGE_H,
              Cfg_InpRawMin := 0,
              Cfg_InpRawMax := 27648,
              Cfg_FailRawHiLim := 29376,
              Cfg_FailRawLoLim := -691,
              Inp_PVBad := false,
              Cfg_FailBypass := false,
              Cfg_FailTripsUnit := true,
              Cfg_FailResetRequired := false,
              Cfg_InFailUsePVEUMax := "AlwaysTRUE",
              Cfg_InFailUsePVEUMin := "AlwaysFALSE",
              Cfg_InFailUseValSub := "AlwaysFALSE",
              Cfg_ValSub := 0.0,
              Cfg_FailDelay := T#0ms,
              Cfg_HasHiHiAlm := "AlwaysTRUE",
              Oset_HiHiLim := "SETTINGS".TT_33303.SP_HH,
              Cfg_HiHiDelay := T#5s,
              Cfg_HiHiDB := 0.0,
              Cfg_HiHiBypass := false,
              Cfg_HiHiTripsUnit := true,
              Cfg_HiHiResetRequired := false,
              Cfg_HasHiAlm := "AlwaysTRUE",
              Oset_HiLim := "SETTINGS".TT_33303.SP_H,
              Cfg_HiDelay := T#5s,
              Cfg_HiDB := 0.0,
              Cfg_HiBypass := false,
              Cfg_HiResetRequired := false,
              Cfg_HasLoAlm := "AlwaysFALSE",
              Oset_LoLim := "SETTINGS".TT_33303.SP_L,
              Cfg_LoDelay := T#5s,
              Cfg_LoDB := 0.0,
              Cfg_LoBypass := false,
              Cfg_LoResetRequired := false,
              Cfg_HasLoLoAlm := "AlwaysFALSE",
              Oset_LoLoLim := "SETTINGS".TT_33303.SP_LL,
              Cfg_LoLoDelay := T#5s,
              Cfg_LoLoDB := 0.0,
              Cfg_LoLoBypass := false,
              Cfg_LoLoTripsUnit := false,
              Cfg_LoLoResetRequired := false,
              Inp_Reset := "RESET",
              PCmd_MOS := false,
              SpareIn1 := 0.0,
              SpareIn2 := 0.0,
              CommonFirstOut := "CMN_FO",
              IsaAlarmFlashing := "UP".ALM_FLASHING,
              IsaTripFlashing := "UP".TRIP_FLASHING);
END_REGION

REGION Network 9: OIL FILTER DIFFERENTIAL PRESSURE
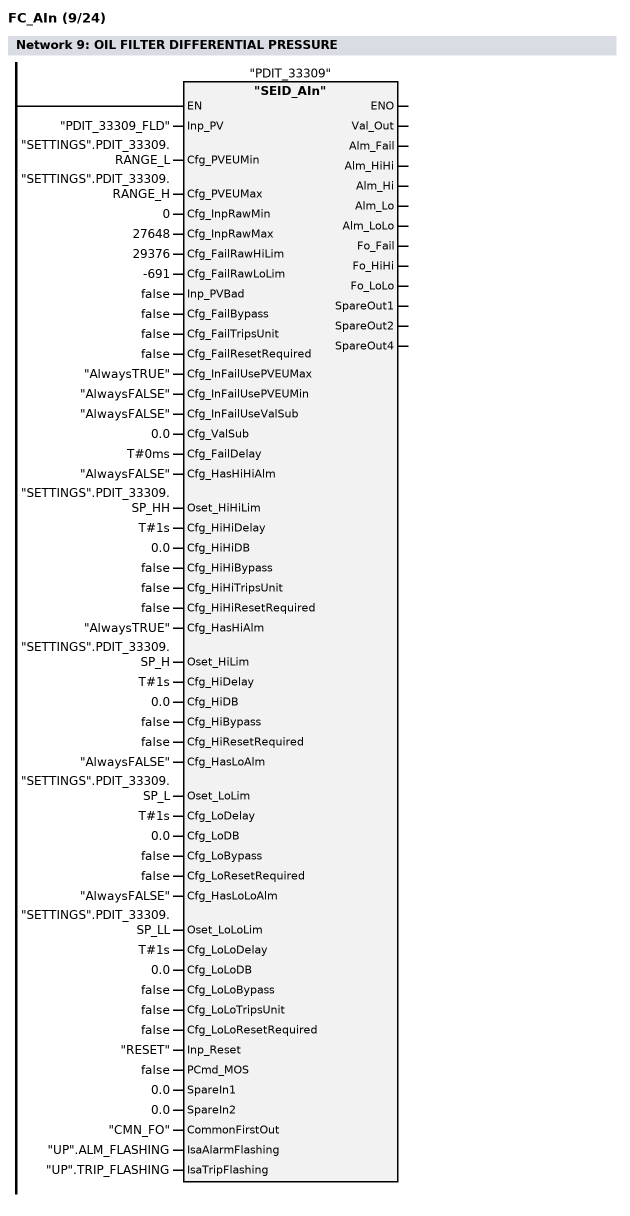
   RUNG wire#powerrail
      "PDIT_33309"(Inp_PV := "PDIT_33309_FLD", Cfg_PVEUMin := "SETTINGS".PDIT_33309.RANGE_L, Cfg_PVEUMax := "SETTINGS".PDIT_33309.RANGE_H, Cfg_InpRawMin := 0, Cfg_InpRawMax := 27648, Cfg_FailRawHiLim := 29376, Cfg_FailRawLoLim := -691, Inp_PVBad := false, Cfg_FailBypass := false, Cfg_FailTripsUnit := false, Cfg_FailResetRequired := false, Cfg_InFailUsePVEUMax := "AlwaysTRUE", Cfg_InFailUsePVEUMin := "AlwaysFALSE", Cfg_InFailUseValSub := "AlwaysFALSE", Cfg_ValSub := 0.0, Cfg_FailDelay := T#0ms, Cfg_HasHiHiAlm := "AlwaysFALSE", Oset_HiHiLim := "SETTINGS".PDIT_33309.SP_HH, Cfg_HiHiDelay := T#1s, Cfg_HiHiDB := 0.0, Cfg_HiHiBypass := false, Cfg_HiHiTripsUnit := false, Cfg_HiHiResetRequired := false, Cfg_HasHiAlm := "AlwaysTRUE", Oset_HiLim := "SETTINGS".PDIT_33309.SP_H, Cfg_HiDelay := T#1s, Cfg_HiDB := 0.0, Cfg_HiBypass := false, Cfg_HiResetRequired := false, Cfg_HasLoAlm := "AlwaysFALSE", Oset_LoLim := "SETTINGS".PDIT_33309.SP_L, Cfg_LoDelay := T#1s, Cfg_LoDB := 0.0, Cfg_LoBypass := false, Cfg_LoResetRequired := false, Cfg_HasLoLoAlm := "AlwaysFALSE", Oset_LoLoLim := "SETTINGS".PDIT_33309.SP_LL, Cfg_LoLoDelay := T#1s, Cfg_LoLoDB := 0.0, Cfg_LoLoBypass := false, Cfg_LoLoTripsUnit := false, Cfg_LoLoResetRequired := false, Inp_Reset := "RESET", PCmd_MOS := false, SpareIn1 := 0.0, SpareIn2 := 0.0, CommonFirstOut := "CMN_FO", IsaAlarmFlashing := "UP".ALM_FLASHING, IsaTripFlashing := "UP".TRIP_FLASHING, Val_Out =>, Alm_Fail =>, Alm_HiHi =>, Alm_Hi =>, Alm_Lo =>, Alm_LoLo =>, Fo_Fail =>, Fo_HiHi =>, Fo_LoLo =>, SpareOut1 =>, SpareOut2 =>, SpareOut4 =>)
   END_RUNG
   // the same network as SCL:
   "PDIT_33309"(Inp_PV := "PDIT_33309_FLD",   // "SEID_AIn"
                Cfg_PVEUMin := "SETTINGS".PDIT_33309.RANGE_L,
                Cfg_PVEUMax := "SETTINGS".PDIT_33309.RANGE_H,
                Cfg_InpRawMin := 0,
                Cfg_InpRawMax := 27648,
                Cfg_FailRawHiLim := 29376,
                Cfg_FailRawLoLim := -691,
                Inp_PVBad := false,
                Cfg_FailBypass := false,
                Cfg_FailTripsUnit := false,
                Cfg_FailResetRequired := false,
                Cfg_InFailUsePVEUMax := "AlwaysTRUE",
                Cfg_InFailUsePVEUMin := "AlwaysFALSE",
                Cfg_InFailUseValSub := "AlwaysFALSE",
                Cfg_ValSub := 0.0,
                Cfg_FailDelay := T#0ms,
                Cfg_HasHiHiAlm := "AlwaysFALSE",
                Oset_HiHiLim := "SETTINGS".PDIT_33309.SP_HH,
                Cfg_HiHiDelay := T#1s,
                Cfg_HiHiDB := 0.0,
                Cfg_HiHiBypass := false,
                Cfg_HiHiTripsUnit := false,
                Cfg_HiHiResetRequired := false,
                Cfg_HasHiAlm := "AlwaysTRUE",
                Oset_HiLim := "SETTINGS".PDIT_33309.SP_H,
                Cfg_HiDelay := T#1s,
                Cfg_HiDB := 0.0,
                Cfg_HiBypass := false,
                Cfg_HiResetRequired := false,
                Cfg_HasLoAlm := "AlwaysFALSE",
                Oset_LoLim := "SETTINGS".PDIT_33309.SP_L,
                Cfg_LoDelay := T#1s,
                Cfg_LoDB := 0.0,
                Cfg_LoBypass := false,
                Cfg_LoResetRequired := false,
                Cfg_HasLoLoAlm := "AlwaysFALSE",
                Oset_LoLoLim := "SETTINGS".PDIT_33309.SP_LL,
                Cfg_LoLoDelay := T#1s,
                Cfg_LoLoDB := 0.0,
                Cfg_LoLoBypass := false,
                Cfg_LoLoTripsUnit := false,
                Cfg_LoLoResetRequired := false,
                Inp_Reset := "RESET",
                PCmd_MOS := false,
                SpareIn1 := 0.0,
                SpareIn2 := 0.0,
                CommonFirstOut := "CMN_FO",
                IsaAlarmFlashing := "UP".ALM_FLASHING,
                IsaTripFlashing := "UP".TRIP_FLASHING);
END_REGION

REGION Network 10: ECONOMIZER PRESSURE
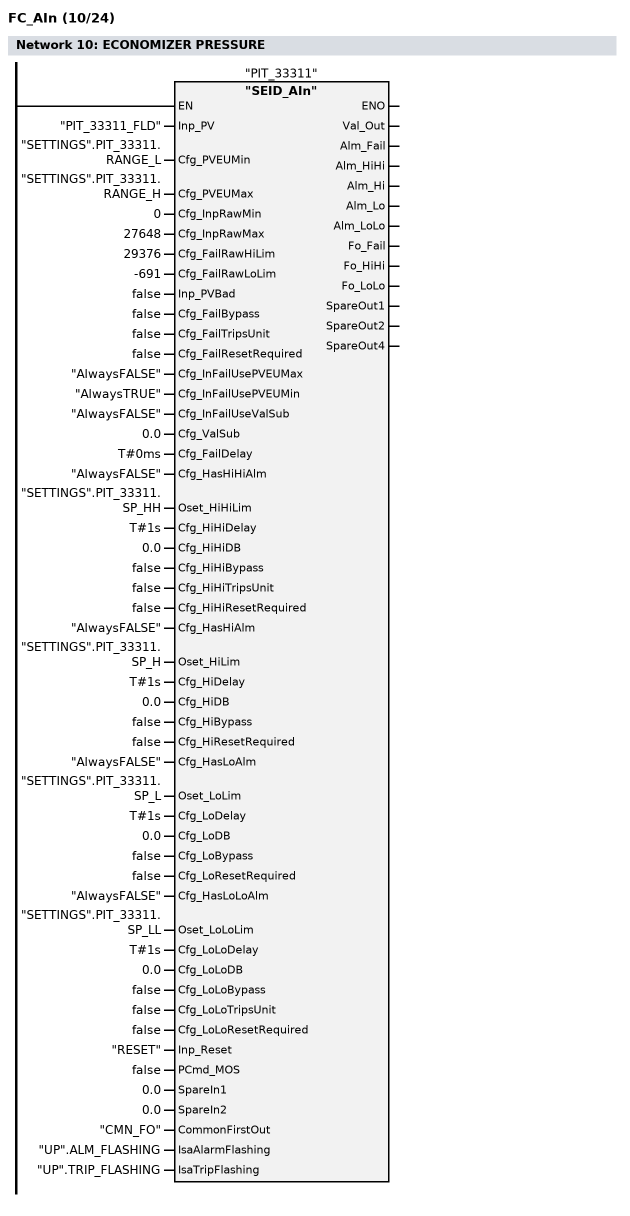
   RUNG wire#powerrail
      "PIT_33311"(Inp_PV := "PIT_33311_FLD", Cfg_PVEUMin := "SETTINGS".PIT_33311.RANGE_L, Cfg_PVEUMax := "SETTINGS".PIT_33311.RANGE_H, Cfg_InpRawMin := 0, Cfg_InpRawMax := 27648, Cfg_FailRawHiLim := 29376, Cfg_FailRawLoLim := -691, Inp_PVBad := false, Cfg_FailBypass := false, Cfg_FailTripsUnit := false, Cfg_FailResetRequired := false, Cfg_InFailUsePVEUMax := "AlwaysFALSE", Cfg_InFailUsePVEUMin := "AlwaysTRUE", Cfg_InFailUseValSub := "AlwaysFALSE", Cfg_ValSub := 0.0, Cfg_FailDelay := T#0ms, Cfg_HasHiHiAlm := "AlwaysFALSE", Oset_HiHiLim := "SETTINGS".PIT_33311.SP_HH, Cfg_HiHiDelay := T#1s, Cfg_HiHiDB := 0.0, Cfg_HiHiBypass := false, Cfg_HiHiTripsUnit := false, Cfg_HiHiResetRequired := false, Cfg_HasHiAlm := "AlwaysFALSE", Oset_HiLim := "SETTINGS".PIT_33311.SP_H, Cfg_HiDelay := T#1s, Cfg_HiDB := 0.0, Cfg_HiBypass := false, Cfg_HiResetRequired := false, Cfg_HasLoAlm := "AlwaysFALSE", Oset_LoLim := "SETTINGS".PIT_33311.SP_L, Cfg_LoDelay := T#1s, Cfg_LoDB := 0.0, Cfg_LoBypass := false, Cfg_LoResetRequired := false, Cfg_HasLoLoAlm := "AlwaysFALSE", Oset_LoLoLim := "SETTINGS".PIT_33311.SP_LL, Cfg_LoLoDelay := T#1s, Cfg_LoLoDB := 0.0, Cfg_LoLoBypass := false, Cfg_LoLoTripsUnit := false, Cfg_LoLoResetRequired := false, Inp_Reset := "RESET", PCmd_MOS := false, SpareIn1 := 0.0, SpareIn2 := 0.0, CommonFirstOut := "CMN_FO", IsaAlarmFlashing := "UP".ALM_FLASHING, IsaTripFlashing := "UP".TRIP_FLASHING, Val_Out =>, Alm_Fail =>, Alm_HiHi =>, Alm_Hi =>, Alm_Lo =>, Alm_LoLo =>, Fo_Fail =>, Fo_HiHi =>, Fo_LoLo =>, SpareOut1 =>, SpareOut2 =>, SpareOut4 =>)
   END_RUNG
   // the same network as SCL:
   "PIT_33311"(Inp_PV := "PIT_33311_FLD",   // "SEID_AIn"
               Cfg_PVEUMin := "SETTINGS".PIT_33311.RANGE_L,
               Cfg_PVEUMax := "SETTINGS".PIT_33311.RANGE_H,
               Cfg_InpRawMin := 0,
               Cfg_InpRawMax := 27648,
               Cfg_FailRawHiLim := 29376,
               Cfg_FailRawLoLim := -691,
               Inp_PVBad := false,
               Cfg_FailBypass := false,
               Cfg_FailTripsUnit := false,
               Cfg_FailResetRequired := false,
               Cfg_InFailUsePVEUMax := "AlwaysFALSE",
               Cfg_InFailUsePVEUMin := "AlwaysTRUE",
               Cfg_InFailUseValSub := "AlwaysFALSE",
               Cfg_ValSub := 0.0,
               Cfg_FailDelay := T#0ms,
               Cfg_HasHiHiAlm := "AlwaysFALSE",
               Oset_HiHiLim := "SETTINGS".PIT_33311.SP_HH,
               Cfg_HiHiDelay := T#1s,
               Cfg_HiHiDB := 0.0,
               Cfg_HiHiBypass := false,
               Cfg_HiHiTripsUnit := false,
               Cfg_HiHiResetRequired := false,
               Cfg_HasHiAlm := "AlwaysFALSE",
               Oset_HiLim := "SETTINGS".PIT_33311.SP_H,
               Cfg_HiDelay := T#1s,
               Cfg_HiDB := 0.0,
               Cfg_HiBypass := false,
               Cfg_HiResetRequired := false,
               Cfg_HasLoAlm := "AlwaysFALSE",
               Oset_LoLim := "SETTINGS".PIT_33311.SP_L,
               Cfg_LoDelay := T#1s,
               Cfg_LoDB := 0.0,
               Cfg_LoBypass := false,
               Cfg_LoResetRequired := false,
               Cfg_HasLoLoAlm := "AlwaysFALSE",
               Oset_LoLoLim := "SETTINGS".PIT_33311.SP_LL,
               Cfg_LoLoDelay := T#1s,
               Cfg_LoLoDB := 0.0,
               Cfg_LoLoBypass := false,
               Cfg_LoLoTripsUnit := false,
               Cfg_LoLoResetRequired := false,
               Inp_Reset := "RESET",
               PCmd_MOS := false,
               SpareIn1 := 0.0,
               SpareIn2 := 0.0,
               CommonFirstOut := "CMN_FO",
               IsaAlarmFlashing := "UP".ALM_FLASHING,
               IsaTripFlashing := "UP".TRIP_FLASHING);
END_REGION

REGION Network 11: ECONOMIZER LEVEL
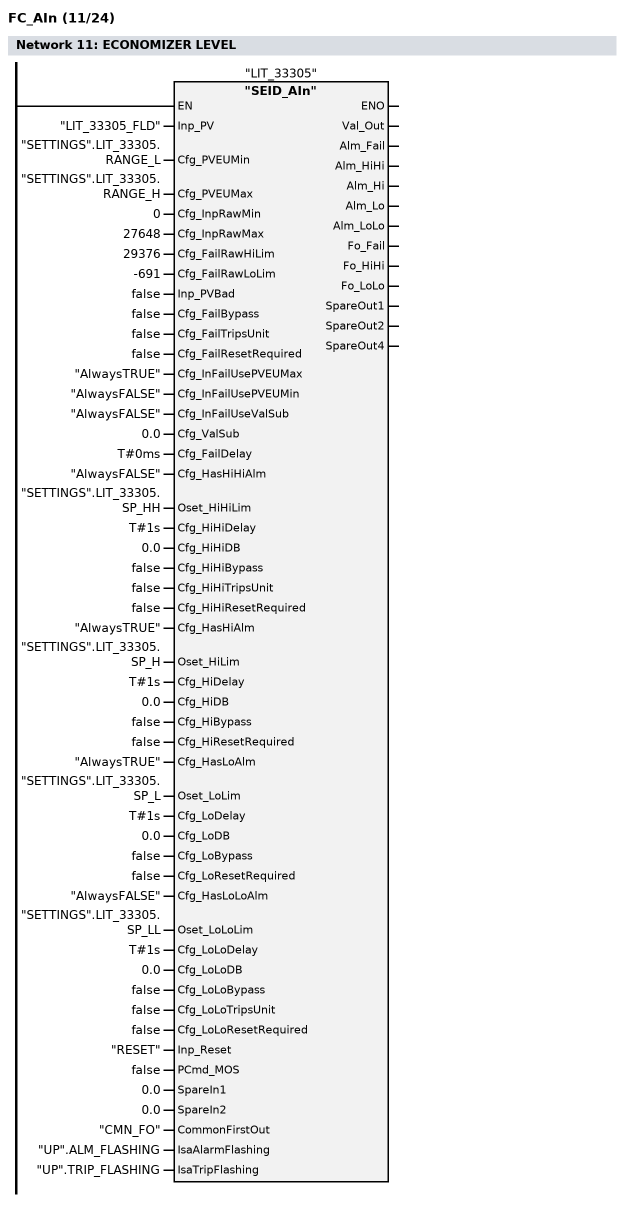
   RUNG wire#powerrail
      "LIT_33305"(Inp_PV := "LIT_33305_FLD", Cfg_PVEUMin := "SETTINGS".LIT_33305.RANGE_L, Cfg_PVEUMax := "SETTINGS".LIT_33305.RANGE_H, Cfg_InpRawMin := 0, Cfg_InpRawMax := 27648, Cfg_FailRawHiLim := 29376, Cfg_FailRawLoLim := -691, Inp_PVBad := false, Cfg_FailBypass := false, Cfg_FailTripsUnit := false, Cfg_FailResetRequired := false, Cfg_InFailUsePVEUMax := "AlwaysTRUE", Cfg_InFailUsePVEUMin := "AlwaysFALSE", Cfg_InFailUseValSub := "AlwaysFALSE", Cfg_ValSub := 0.0, Cfg_FailDelay := T#0ms, Cfg_HasHiHiAlm := "AlwaysFALSE", Oset_HiHiLim := "SETTINGS".LIT_33305.SP_HH, Cfg_HiHiDelay := T#1s, Cfg_HiHiDB := 0.0, Cfg_HiHiBypass := false, Cfg_HiHiTripsUnit := false, Cfg_HiHiResetRequired := false, Cfg_HasHiAlm := "AlwaysTRUE", Oset_HiLim := "SETTINGS".LIT_33305.SP_H, Cfg_HiDelay := T#1s, Cfg_HiDB := 0.0, Cfg_HiBypass := false, Cfg_HiResetRequired := false, Cfg_HasLoAlm := "AlwaysTRUE", Oset_LoLim := "SETTINGS".LIT_33305.SP_L, Cfg_LoDelay := T#1s, Cfg_LoDB := 0.0, Cfg_LoBypass := false, Cfg_LoResetRequired := false, Cfg_HasLoLoAlm := "AlwaysFALSE", Oset_LoLoLim := "SETTINGS".LIT_33305.SP_LL, Cfg_LoLoDelay := T#1s, Cfg_LoLoDB := 0.0, Cfg_LoLoBypass := false, Cfg_LoLoTripsUnit := false, Cfg_LoLoResetRequired := false, Inp_Reset := "RESET", PCmd_MOS := false, SpareIn1 := 0.0, SpareIn2 := 0.0, CommonFirstOut := "CMN_FO", IsaAlarmFlashing := "UP".ALM_FLASHING, IsaTripFlashing := "UP".TRIP_FLASHING, Val_Out =>, Alm_Fail =>, Alm_HiHi =>, Alm_Hi =>, Alm_Lo =>, Alm_LoLo =>, Fo_Fail =>, Fo_HiHi =>, Fo_LoLo =>, SpareOut1 =>, SpareOut2 =>, SpareOut4 =>)
   END_RUNG
   // the same network as SCL:
   "LIT_33305"(Inp_PV := "LIT_33305_FLD",   // "SEID_AIn"
               Cfg_PVEUMin := "SETTINGS".LIT_33305.RANGE_L,
               Cfg_PVEUMax := "SETTINGS".LIT_33305.RANGE_H,
               Cfg_InpRawMin := 0,
               Cfg_InpRawMax := 27648,
               Cfg_FailRawHiLim := 29376,
               Cfg_FailRawLoLim := -691,
               Inp_PVBad := false,
               Cfg_FailBypass := false,
               Cfg_FailTripsUnit := false,
               Cfg_FailResetRequired := false,
               Cfg_InFailUsePVEUMax := "AlwaysTRUE",
               Cfg_InFailUsePVEUMin := "AlwaysFALSE",
               Cfg_InFailUseValSub := "AlwaysFALSE",
               Cfg_ValSub := 0.0,
               Cfg_FailDelay := T#0ms,
               Cfg_HasHiHiAlm := "AlwaysFALSE",
               Oset_HiHiLim := "SETTINGS".LIT_33305.SP_HH,
               Cfg_HiHiDelay := T#1s,
               Cfg_HiHiDB := 0.0,
               Cfg_HiHiBypass := false,
               Cfg_HiHiTripsUnit := false,
               Cfg_HiHiResetRequired := false,
               Cfg_HasHiAlm := "AlwaysTRUE",
               Oset_HiLim := "SETTINGS".LIT_33305.SP_H,
               Cfg_HiDelay := T#1s,
               Cfg_HiDB := 0.0,
               Cfg_HiBypass := false,
               Cfg_HiResetRequired := false,
               Cfg_HasLoAlm := "AlwaysTRUE",
               Oset_LoLim := "SETTINGS".LIT_33305.SP_L,
               Cfg_LoDelay := T#1s,
               Cfg_LoDB := 0.0,
               Cfg_LoBypass := false,
               Cfg_LoResetRequired := false,
               Cfg_HasLoLoAlm := "AlwaysFALSE",
               Oset_LoLoLim := "SETTINGS".LIT_33305.SP_LL,
               Cfg_LoLoDelay := T#1s,
               Cfg_LoLoDB := 0.0,
               Cfg_LoLoBypass := false,
               Cfg_LoLoTripsUnit := false,
               Cfg_LoLoResetRequired := false,
               Inp_Reset := "RESET",
               PCmd_MOS := false,
               SpareIn1 := 0.0,
               SpareIn2 := 0.0,
               CommonFirstOut := "CMN_FO",
               IsaAlarmFlashing := "UP".ALM_FLASHING,
               IsaTripFlashing := "UP".TRIP_FLASHING);
END_REGION

REGION Network 12: KO DRUM LEVEL
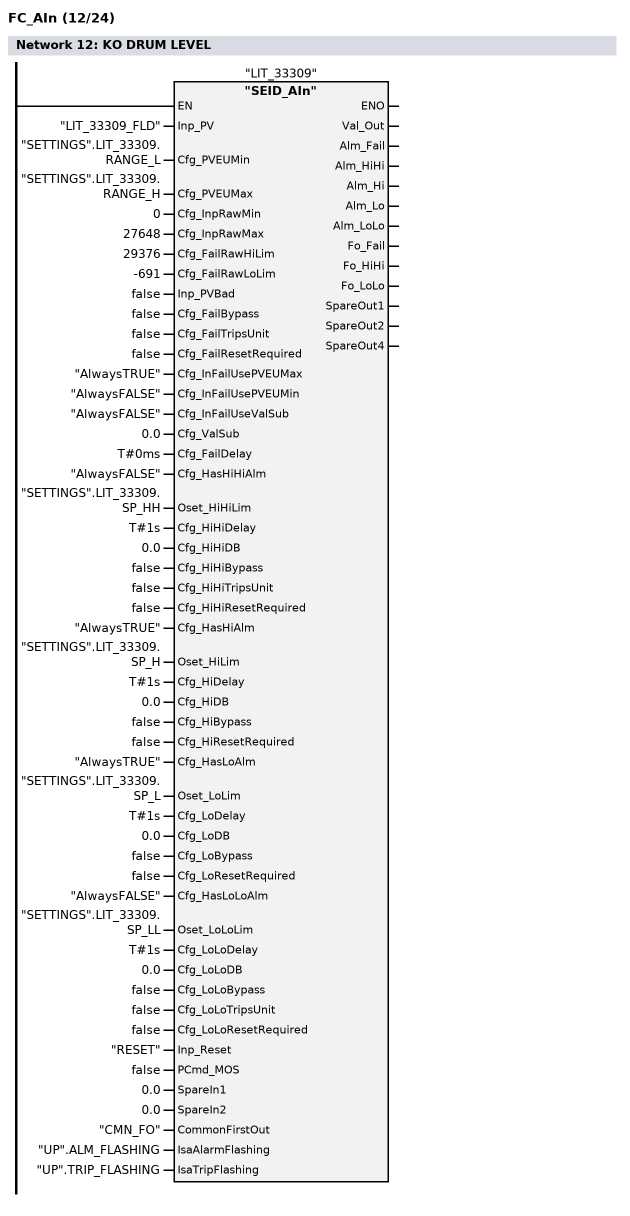
   RUNG wire#powerrail
      "LIT_33309"(Inp_PV := "LIT_33309_FLD", Cfg_PVEUMin := "SETTINGS".LIT_33309.RANGE_L, Cfg_PVEUMax := "SETTINGS".LIT_33309.RANGE_H, Cfg_InpRawMin := 0, Cfg_InpRawMax := 27648, Cfg_FailRawHiLim := 29376, Cfg_FailRawLoLim := -691, Inp_PVBad := false, Cfg_FailBypass := false, Cfg_FailTripsUnit := false, Cfg_FailResetRequired := false, Cfg_InFailUsePVEUMax := "AlwaysTRUE", Cfg_InFailUsePVEUMin := "AlwaysFALSE", Cfg_InFailUseValSub := "AlwaysFALSE", Cfg_ValSub := 0.0, Cfg_FailDelay := T#0ms, Cfg_HasHiHiAlm := "AlwaysFALSE", Oset_HiHiLim := "SETTINGS".LIT_33309.SP_HH, Cfg_HiHiDelay := T#1s, Cfg_HiHiDB := 0.0, Cfg_HiHiBypass := false, Cfg_HiHiTripsUnit := false, Cfg_HiHiResetRequired := false, Cfg_HasHiAlm := "AlwaysTRUE", Oset_HiLim := "SETTINGS".LIT_33309.SP_H, Cfg_HiDelay := T#1s, Cfg_HiDB := 0.0, Cfg_HiBypass := false, Cfg_HiResetRequired := false, Cfg_HasLoAlm := "AlwaysTRUE", Oset_LoLim := "SETTINGS".LIT_33309.SP_L, Cfg_LoDelay := T#1s, Cfg_LoDB := 0.0, Cfg_LoBypass := false, Cfg_LoResetRequired := false, Cfg_HasLoLoAlm := "AlwaysFALSE", Oset_LoLoLim := "SETTINGS".LIT_33309.SP_LL, Cfg_LoLoDelay := T#1s, Cfg_LoLoDB := 0.0, Cfg_LoLoBypass := false, Cfg_LoLoTripsUnit := false, Cfg_LoLoResetRequired := false, Inp_Reset := "RESET", PCmd_MOS := false, SpareIn1 := 0.0, SpareIn2 := 0.0, CommonFirstOut := "CMN_FO", IsaAlarmFlashing := "UP".ALM_FLASHING, IsaTripFlashing := "UP".TRIP_FLASHING, Val_Out =>, Alm_Fail =>, Alm_HiHi =>, Alm_Hi =>, Alm_Lo =>, Alm_LoLo =>, Fo_Fail =>, Fo_HiHi =>, Fo_LoLo =>, SpareOut1 =>, SpareOut2 =>, SpareOut4 =>)
   END_RUNG
   // the same network as SCL:
   "LIT_33309"(Inp_PV := "LIT_33309_FLD",   // "SEID_AIn"
               Cfg_PVEUMin := "SETTINGS".LIT_33309.RANGE_L,
               Cfg_PVEUMax := "SETTINGS".LIT_33309.RANGE_H,
               Cfg_InpRawMin := 0,
               Cfg_InpRawMax := 27648,
               Cfg_FailRawHiLim := 29376,
               Cfg_FailRawLoLim := -691,
               Inp_PVBad := false,
               Cfg_FailBypass := false,
               Cfg_FailTripsUnit := false,
               Cfg_FailResetRequired := false,
               Cfg_InFailUsePVEUMax := "AlwaysTRUE",
               Cfg_InFailUsePVEUMin := "AlwaysFALSE",
               Cfg_InFailUseValSub := "AlwaysFALSE",
               Cfg_ValSub := 0.0,
               Cfg_FailDelay := T#0ms,
               Cfg_HasHiHiAlm := "AlwaysFALSE",
               Oset_HiHiLim := "SETTINGS".LIT_33309.SP_HH,
               Cfg_HiHiDelay := T#1s,
               Cfg_HiHiDB := 0.0,
               Cfg_HiHiBypass := false,
               Cfg_HiHiTripsUnit := false,
               Cfg_HiHiResetRequired := false,
               Cfg_HasHiAlm := "AlwaysTRUE",
               Oset_HiLim := "SETTINGS".LIT_33309.SP_H,
               Cfg_HiDelay := T#1s,
               Cfg_HiDB := 0.0,
               Cfg_HiBypass := false,
               Cfg_HiResetRequired := false,
               Cfg_HasLoAlm := "AlwaysTRUE",
               Oset_LoLim := "SETTINGS".LIT_33309.SP_L,
               Cfg_LoDelay := T#1s,
               Cfg_LoDB := 0.0,
               Cfg_LoBypass := false,
               Cfg_LoResetRequired := false,
               Cfg_HasLoLoAlm := "AlwaysFALSE",
               Oset_LoLoLim := "SETTINGS".LIT_33309.SP_LL,
               Cfg_LoLoDelay := T#1s,
               Cfg_LoLoDB := 0.0,
               Cfg_LoLoBypass := false,
               Cfg_LoLoTripsUnit := false,
               Cfg_LoLoResetRequired := false,
               Inp_Reset := "RESET",
               PCmd_MOS := false,
               SpareIn1 := 0.0,
               SpareIn2 := 0.0,
               CommonFirstOut := "CMN_FO",
               IsaAlarmFlashing := "UP".ALM_FLASHING,
               IsaTripFlashing := "UP".TRIP_FLASHING);
END_REGION

REGION Network 13: LUBE OIL RECOVERY LINE PRESSURE
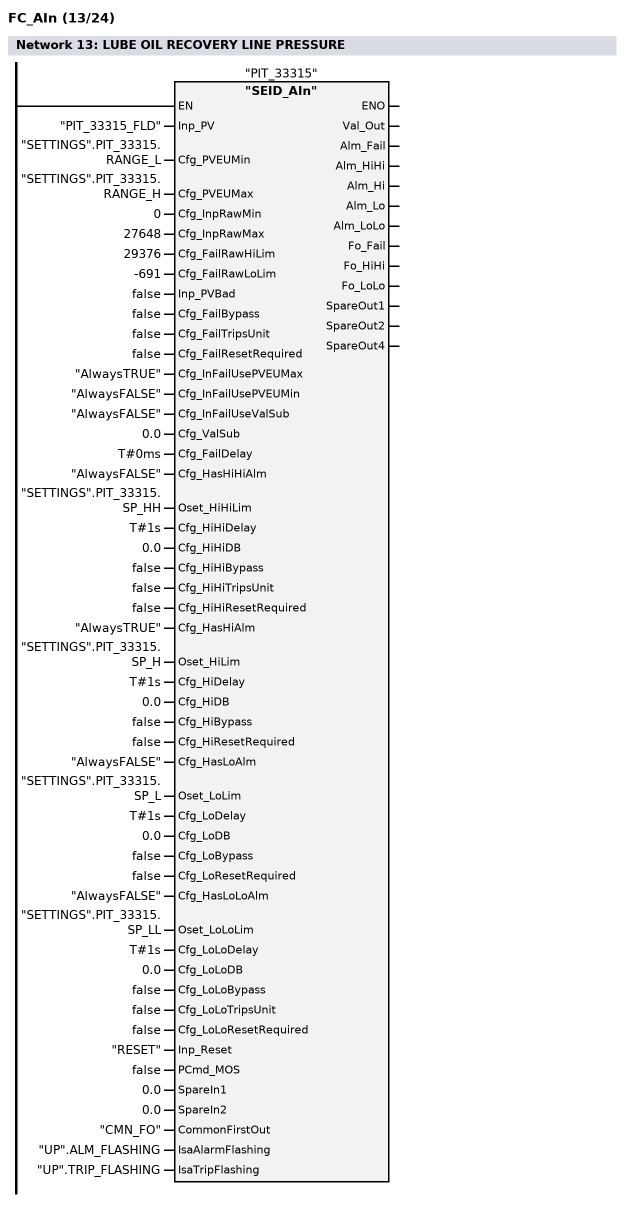
   RUNG wire#powerrail
      "PIT_33315"(Inp_PV := "PIT_33315_FLD", Cfg_PVEUMin := "SETTINGS".PIT_33315.RANGE_L, Cfg_PVEUMax := "SETTINGS".PIT_33315.RANGE_H, Cfg_InpRawMin := 0, Cfg_InpRawMax := 27648, Cfg_FailRawHiLim := 29376, Cfg_FailRawLoLim := -691, Inp_PVBad := false, Cfg_FailBypass := false, Cfg_FailTripsUnit := false, Cfg_FailResetRequired := false, Cfg_InFailUsePVEUMax := "AlwaysTRUE", Cfg_InFailUsePVEUMin := "AlwaysFALSE", Cfg_InFailUseValSub := "AlwaysFALSE", Cfg_ValSub := 0.0, Cfg_FailDelay := T#0ms, Cfg_HasHiHiAlm := "AlwaysFALSE", Oset_HiHiLim := "SETTINGS".PIT_33315.SP_HH, Cfg_HiHiDelay := T#1s, Cfg_HiHiDB := 0.0, Cfg_HiHiBypass := false, Cfg_HiHiTripsUnit := false, Cfg_HiHiResetRequired := false, Cfg_HasHiAlm := "AlwaysTRUE", Oset_HiLim := "SETTINGS".PIT_33315.SP_H, Cfg_HiDelay := T#1s, Cfg_HiDB := 0.0, Cfg_HiBypass := false, Cfg_HiResetRequired := false, Cfg_HasLoAlm := "AlwaysFALSE", Oset_LoLim := "SETTINGS".PIT_33315.SP_L, Cfg_LoDelay := T#1s, Cfg_LoDB := 0.0, Cfg_LoBypass := false, Cfg_LoResetRequired := false, Cfg_HasLoLoAlm := "AlwaysFALSE", Oset_LoLoLim := "SETTINGS".PIT_33315.SP_LL, Cfg_LoLoDelay := T#1s, Cfg_LoLoDB := 0.0, Cfg_LoLoBypass := false, Cfg_LoLoTripsUnit := false, Cfg_LoLoResetRequired := false, Inp_Reset := "RESET", PCmd_MOS := false, SpareIn1 := 0.0, SpareIn2 := 0.0, CommonFirstOut := "CMN_FO", IsaAlarmFlashing := "UP".ALM_FLASHING, IsaTripFlashing := "UP".TRIP_FLASHING, Val_Out =>, Alm_Fail =>, Alm_HiHi =>, Alm_Hi =>, Alm_Lo =>, Alm_LoLo =>, Fo_Fail =>, Fo_HiHi =>, Fo_LoLo =>, SpareOut1 =>, SpareOut2 =>, SpareOut4 =>)
   END_RUNG
   // the same network as SCL:
   "PIT_33315"(Inp_PV := "PIT_33315_FLD",   // "SEID_AIn"
               Cfg_PVEUMin := "SETTINGS".PIT_33315.RANGE_L,
               Cfg_PVEUMax := "SETTINGS".PIT_33315.RANGE_H,
               Cfg_InpRawMin := 0,
               Cfg_InpRawMax := 27648,
               Cfg_FailRawHiLim := 29376,
               Cfg_FailRawLoLim := -691,
               Inp_PVBad := false,
               Cfg_FailBypass := false,
               Cfg_FailTripsUnit := false,
               Cfg_FailResetRequired := false,
               Cfg_InFailUsePVEUMax := "AlwaysTRUE",
               Cfg_InFailUsePVEUMin := "AlwaysFALSE",
               Cfg_InFailUseValSub := "AlwaysFALSE",
               Cfg_ValSub := 0.0,
               Cfg_FailDelay := T#0ms,
               Cfg_HasHiHiAlm := "AlwaysFALSE",
               Oset_HiHiLim := "SETTINGS".PIT_33315.SP_HH,
               Cfg_HiHiDelay := T#1s,
               Cfg_HiHiDB := 0.0,
               Cfg_HiHiBypass := false,
               Cfg_HiHiTripsUnit := false,
               Cfg_HiHiResetRequired := false,
               Cfg_HasHiAlm := "AlwaysTRUE",
               Oset_HiLim := "SETTINGS".PIT_33315.SP_H,
               Cfg_HiDelay := T#1s,
               Cfg_HiDB := 0.0,
               Cfg_HiBypass := false,
               Cfg_HiResetRequired := false,
               Cfg_HasLoAlm := "AlwaysFALSE",
               Oset_LoLim := "SETTINGS".PIT_33315.SP_L,
               Cfg_LoDelay := T#1s,
               Cfg_LoDB := 0.0,
               Cfg_LoBypass := false,
               Cfg_LoResetRequired := false,
               Cfg_HasLoLoAlm := "AlwaysFALSE",
               Oset_LoLoLim := "SETTINGS".PIT_33315.SP_LL,
               Cfg_LoLoDelay := T#1s,
               Cfg_LoLoDB := 0.0,
               Cfg_LoLoBypass := false,
               Cfg_LoLoTripsUnit := false,
               Cfg_LoLoResetRequired := false,
               Inp_Reset := "RESET",
               PCmd_MOS := false,
               SpareIn1 := 0.0,
               SpareIn2 := 0.0,
               CommonFirstOut := "CMN_FO",
               IsaAlarmFlashing := "UP".ALM_FLASHING,
               IsaTripFlashing := "UP".TRIP_FLASHING);
END_REGION

REGION Network 14: OIL SEPARATOR LEVEL
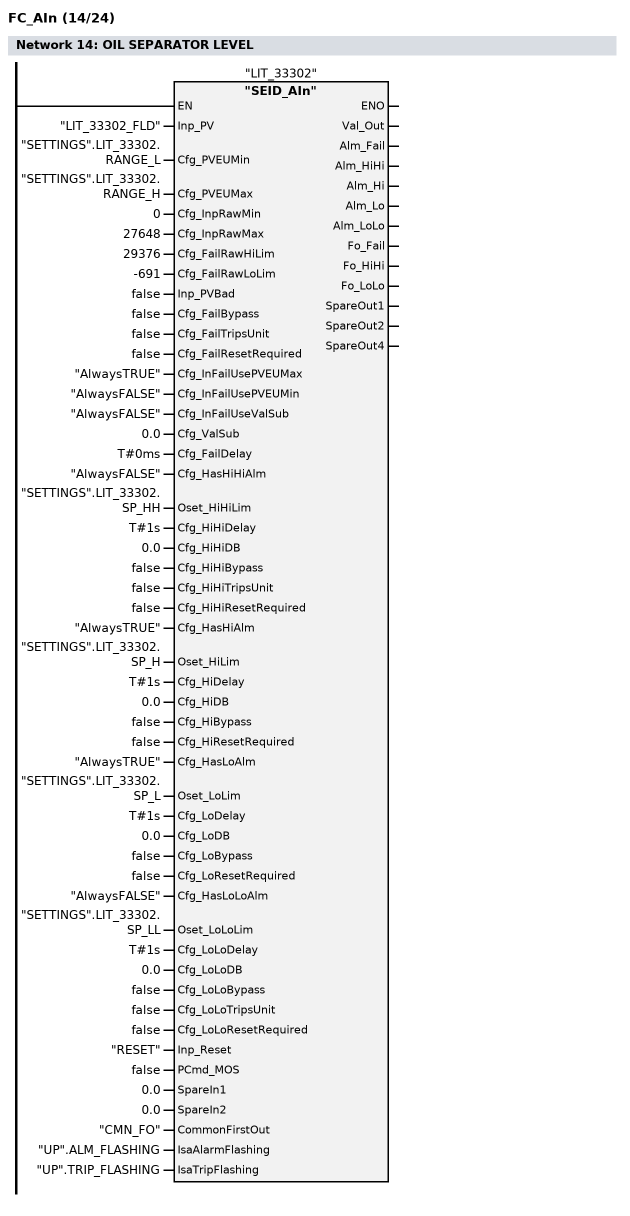
   RUNG wire#powerrail
      "LIT_33302"(Inp_PV := "LIT_33302_FLD", Cfg_PVEUMin := "SETTINGS".LIT_33302.RANGE_L, Cfg_PVEUMax := "SETTINGS".LIT_33302.RANGE_H, Cfg_InpRawMin := 0, Cfg_InpRawMax := 27648, Cfg_FailRawHiLim := 29376, Cfg_FailRawLoLim := -691, Inp_PVBad := false, Cfg_FailBypass := false, Cfg_FailTripsUnit := false, Cfg_FailResetRequired := false, Cfg_InFailUsePVEUMax := "AlwaysTRUE", Cfg_InFailUsePVEUMin := "AlwaysFALSE", Cfg_InFailUseValSub := "AlwaysFALSE", Cfg_ValSub := 0.0, Cfg_FailDelay := T#0ms, Cfg_HasHiHiAlm := "AlwaysFALSE", Oset_HiHiLim := "SETTINGS".LIT_33302.SP_HH, Cfg_HiHiDelay := T#1s, Cfg_HiHiDB := 0.0, Cfg_HiHiBypass := false, Cfg_HiHiTripsUnit := false, Cfg_HiHiResetRequired := false, Cfg_HasHiAlm := "AlwaysTRUE", Oset_HiLim := "SETTINGS".LIT_33302.SP_H, Cfg_HiDelay := T#1s, Cfg_HiDB := 0.0, Cfg_HiBypass := false, Cfg_HiResetRequired := false, Cfg_HasLoAlm := "AlwaysTRUE", Oset_LoLim := "SETTINGS".LIT_33302.SP_L, Cfg_LoDelay := T#1s, Cfg_LoDB := 0.0, Cfg_LoBypass := false, Cfg_LoResetRequired := false, Cfg_HasLoLoAlm := "AlwaysFALSE", Oset_LoLoLim := "SETTINGS".LIT_33302.SP_LL, Cfg_LoLoDelay := T#1s, Cfg_LoLoDB := 0.0, Cfg_LoLoBypass := false, Cfg_LoLoTripsUnit := false, Cfg_LoLoResetRequired := false, Inp_Reset := "RESET", PCmd_MOS := false, SpareIn1 := 0.0, SpareIn2 := 0.0, CommonFirstOut := "CMN_FO", IsaAlarmFlashing := "UP".ALM_FLASHING, IsaTripFlashing := "UP".TRIP_FLASHING, Val_Out =>, Alm_Fail =>, Alm_HiHi =>, Alm_Hi =>, Alm_Lo =>, Alm_LoLo =>, Fo_Fail =>, Fo_HiHi =>, Fo_LoLo =>, SpareOut1 =>, SpareOut2 =>, SpareOut4 =>)
   END_RUNG
   // the same network as SCL:
   "LIT_33302"(Inp_PV := "LIT_33302_FLD",   // "SEID_AIn"
               Cfg_PVEUMin := "SETTINGS".LIT_33302.RANGE_L,
               Cfg_PVEUMax := "SETTINGS".LIT_33302.RANGE_H,
               Cfg_InpRawMin := 0,
               Cfg_InpRawMax := 27648,
               Cfg_FailRawHiLim := 29376,
               Cfg_FailRawLoLim := -691,
               Inp_PVBad := false,
               Cfg_FailBypass := false,
               Cfg_FailTripsUnit := false,
               Cfg_FailResetRequired := false,
               Cfg_InFailUsePVEUMax := "AlwaysTRUE",
               Cfg_InFailUsePVEUMin := "AlwaysFALSE",
               Cfg_InFailUseValSub := "AlwaysFALSE",
               Cfg_ValSub := 0.0,
               Cfg_FailDelay := T#0ms,
               Cfg_HasHiHiAlm := "AlwaysFALSE",
               Oset_HiHiLim := "SETTINGS".LIT_33302.SP_HH,
               Cfg_HiHiDelay := T#1s,
               Cfg_HiHiDB := 0.0,
               Cfg_HiHiBypass := false,
               Cfg_HiHiTripsUnit := false,
               Cfg_HiHiResetRequired := false,
               Cfg_HasHiAlm := "AlwaysTRUE",
               Oset_HiLim := "SETTINGS".LIT_33302.SP_H,
               Cfg_HiDelay := T#1s,
               Cfg_HiDB := 0.0,
               Cfg_HiBypass := false,
               Cfg_HiResetRequired := false,
               Cfg_HasLoAlm := "AlwaysTRUE",
               Oset_LoLim := "SETTINGS".LIT_33302.SP_L,
               Cfg_LoDelay := T#1s,
               Cfg_LoDB := 0.0,
               Cfg_LoBypass := false,
               Cfg_LoResetRequired := false,
               Cfg_HasLoLoAlm := "AlwaysFALSE",
               Oset_LoLoLim := "SETTINGS".LIT_33302.SP_LL,
               Cfg_LoLoDelay := T#1s,
               Cfg_LoLoDB := 0.0,
               Cfg_LoLoBypass := false,
               Cfg_LoLoTripsUnit := false,
               Cfg_LoLoResetRequired := false,
               Inp_Reset := "RESET",
               PCmd_MOS := false,
               SpareIn1 := 0.0,
               SpareIn2 := 0.0,
               CommonFirstOut := "CMN_FO",
               IsaAlarmFlashing := "UP".ALM_FLASHING,
               IsaTripFlashing := "UP".TRIP_FLASHING);
END_REGION

REGION Network 15: SEAL NITROGEN FLOW
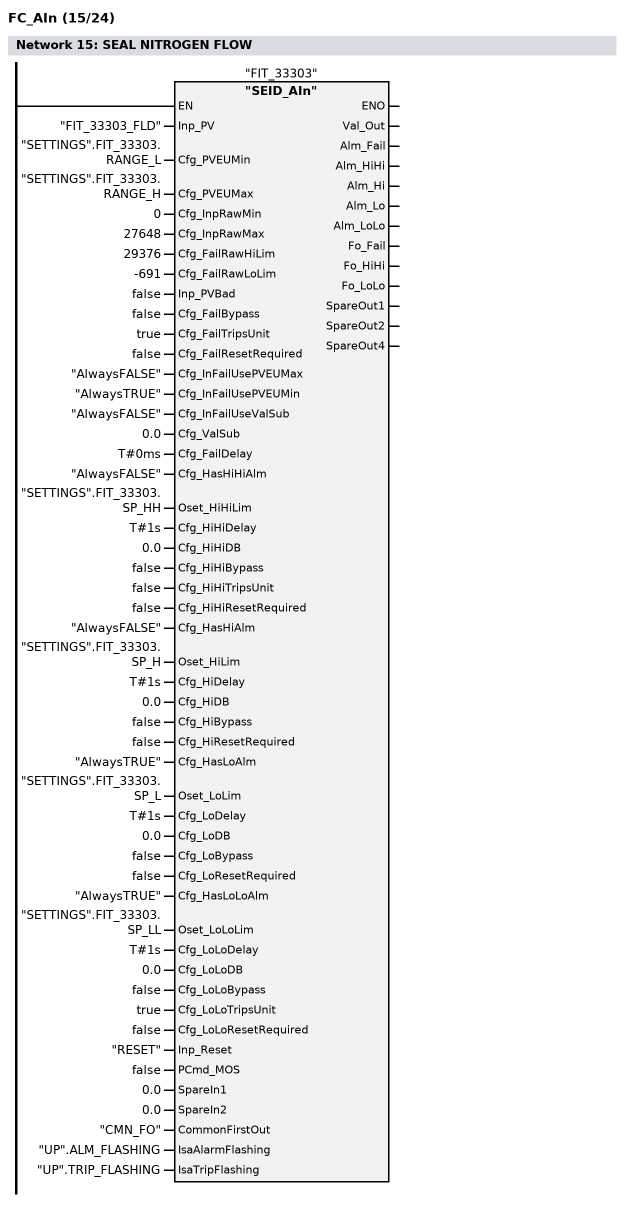
   RUNG wire#powerrail
      "FIT_33303"(Inp_PV := "FIT_33303_FLD", Cfg_PVEUMin := "SETTINGS".FIT_33303.RANGE_L, Cfg_PVEUMax := "SETTINGS".FIT_33303.RANGE_H, Cfg_InpRawMin := 0, Cfg_InpRawMax := 27648, Cfg_FailRawHiLim := 29376, Cfg_FailRawLoLim := -691, Inp_PVBad := false, Cfg_FailBypass := false, Cfg_FailTripsUnit := true, Cfg_FailResetRequired := false, Cfg_InFailUsePVEUMax := "AlwaysFALSE", Cfg_InFailUsePVEUMin := "AlwaysTRUE", Cfg_InFailUseValSub := "AlwaysFALSE", Cfg_ValSub := 0.0, Cfg_FailDelay := T#0ms, Cfg_HasHiHiAlm := "AlwaysFALSE", Oset_HiHiLim := "SETTINGS".FIT_33303.SP_HH, Cfg_HiHiDelay := T#1s, Cfg_HiHiDB := 0.0, Cfg_HiHiBypass := false, Cfg_HiHiTripsUnit := false, Cfg_HiHiResetRequired := false, Cfg_HasHiAlm := "AlwaysFALSE", Oset_HiLim := "SETTINGS".FIT_33303.SP_H, Cfg_HiDelay := T#1s, Cfg_HiDB := 0.0, Cfg_HiBypass := false, Cfg_HiResetRequired := false, Cfg_HasLoAlm := "AlwaysTRUE", Oset_LoLim := "SETTINGS".FIT_33303.SP_L, Cfg_LoDelay := T#1s, Cfg_LoDB := 0.0, Cfg_LoBypass := false, Cfg_LoResetRequired := false, Cfg_HasLoLoAlm := "AlwaysTRUE", Oset_LoLoLim := "SETTINGS".FIT_33303.SP_LL, Cfg_LoLoDelay := T#1s, Cfg_LoLoDB := 0.0, Cfg_LoLoBypass := false, Cfg_LoLoTripsUnit := true, Cfg_LoLoResetRequired := false, Inp_Reset := "RESET", PCmd_MOS := false, SpareIn1 := 0.0, SpareIn2 := 0.0, CommonFirstOut := "CMN_FO", IsaAlarmFlashing := "UP".ALM_FLASHING, IsaTripFlashing := "UP".TRIP_FLASHING, Val_Out =>, Alm_Fail =>, Alm_HiHi =>, Alm_Hi =>, Alm_Lo =>, Alm_LoLo =>, Fo_Fail =>, Fo_HiHi =>, Fo_LoLo =>, SpareOut1 =>, SpareOut2 =>, SpareOut4 =>)
   END_RUNG
   // the same network as SCL:
   "FIT_33303"(Inp_PV := "FIT_33303_FLD",   // "SEID_AIn"
               Cfg_PVEUMin := "SETTINGS".FIT_33303.RANGE_L,
               Cfg_PVEUMax := "SETTINGS".FIT_33303.RANGE_H,
               Cfg_InpRawMin := 0,
               Cfg_InpRawMax := 27648,
               Cfg_FailRawHiLim := 29376,
               Cfg_FailRawLoLim := -691,
               Inp_PVBad := false,
               Cfg_FailBypass := false,
               Cfg_FailTripsUnit := true,
               Cfg_FailResetRequired := false,
               Cfg_InFailUsePVEUMax := "AlwaysFALSE",
               Cfg_InFailUsePVEUMin := "AlwaysTRUE",
               Cfg_InFailUseValSub := "AlwaysFALSE",
               Cfg_ValSub := 0.0,
               Cfg_FailDelay := T#0ms,
               Cfg_HasHiHiAlm := "AlwaysFALSE",
               Oset_HiHiLim := "SETTINGS".FIT_33303.SP_HH,
               Cfg_HiHiDelay := T#1s,
               Cfg_HiHiDB := 0.0,
               Cfg_HiHiBypass := false,
               Cfg_HiHiTripsUnit := false,
               Cfg_HiHiResetRequired := false,
               Cfg_HasHiAlm := "AlwaysFALSE",
               Oset_HiLim := "SETTINGS".FIT_33303.SP_H,
               Cfg_HiDelay := T#1s,
               Cfg_HiDB := 0.0,
               Cfg_HiBypass := false,
               Cfg_HiResetRequired := false,
               Cfg_HasLoAlm := "AlwaysTRUE",
               Oset_LoLim := "SETTINGS".FIT_33303.SP_L,
               Cfg_LoDelay := T#1s,
               Cfg_LoDB := 0.0,
               Cfg_LoBypass := false,
               Cfg_LoResetRequired := false,
               Cfg_HasLoLoAlm := "AlwaysTRUE",
               Oset_LoLoLim := "SETTINGS".FIT_33303.SP_LL,
               Cfg_LoLoDelay := T#1s,
               Cfg_LoLoDB := 0.0,
               Cfg_LoLoBypass := false,
               Cfg_LoLoTripsUnit := true,
               Cfg_LoLoResetRequired := false,
               Inp_Reset := "RESET",
               PCmd_MOS := false,
               SpareIn1 := 0.0,
               SpareIn2 := 0.0,
               CommonFirstOut := "CMN_FO",
               IsaAlarmFlashing := "UP".ALM_FLASHING,
               IsaTripFlashing := "UP".TRIP_FLASHING);
END_REGION

REGION Network 16: COMPRESSOR SEAL POT LEVEL
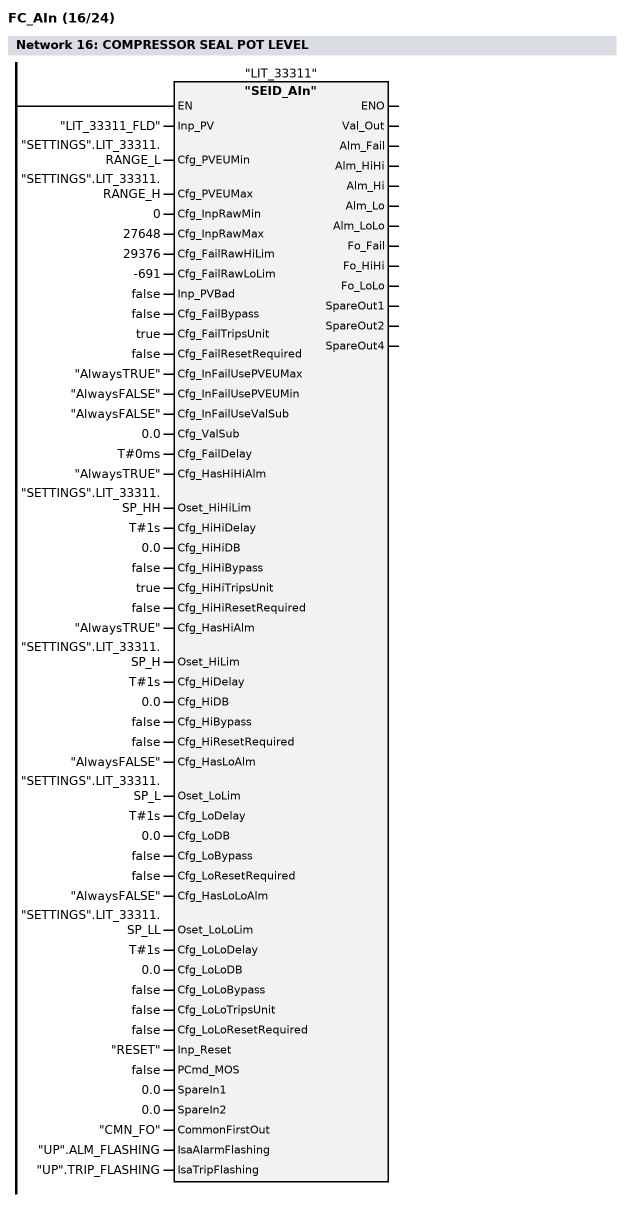
   RUNG wire#powerrail
      "LIT_33311"(Inp_PV := "LIT_33311_FLD", Cfg_PVEUMin := "SETTINGS".LIT_33311.RANGE_L, Cfg_PVEUMax := "SETTINGS".LIT_33311.RANGE_H, Cfg_InpRawMin := 0, Cfg_InpRawMax := 27648, Cfg_FailRawHiLim := 29376, Cfg_FailRawLoLim := -691, Inp_PVBad := false, Cfg_FailBypass := false, Cfg_FailTripsUnit := true, Cfg_FailResetRequired := false, Cfg_InFailUsePVEUMax := "AlwaysTRUE", Cfg_InFailUsePVEUMin := "AlwaysFALSE", Cfg_InFailUseValSub := "AlwaysFALSE", Cfg_ValSub := 0.0, Cfg_FailDelay := T#0ms, Cfg_HasHiHiAlm := "AlwaysTRUE", Oset_HiHiLim := "SETTINGS".LIT_33311.SP_HH, Cfg_HiHiDelay := T#1s, Cfg_HiHiDB := 0.0, Cfg_HiHiBypass := false, Cfg_HiHiTripsUnit := true, Cfg_HiHiResetRequired := false, Cfg_HasHiAlm := "AlwaysTRUE", Oset_HiLim := "SETTINGS".LIT_33311.SP_H, Cfg_HiDelay := T#1s, Cfg_HiDB := 0.0, Cfg_HiBypass := false, Cfg_HiResetRequired := false, Cfg_HasLoAlm := "AlwaysFALSE", Oset_LoLim := "SETTINGS".LIT_33311.SP_L, Cfg_LoDelay := T#1s, Cfg_LoDB := 0.0, Cfg_LoBypass := false, Cfg_LoResetRequired := false, Cfg_HasLoLoAlm := "AlwaysFALSE", Oset_LoLoLim := "SETTINGS".LIT_33311.SP_LL, Cfg_LoLoDelay := T#1s, Cfg_LoLoDB := 0.0, Cfg_LoLoBypass := false, Cfg_LoLoTripsUnit := false, Cfg_LoLoResetRequired := false, Inp_Reset := "RESET", PCmd_MOS := false, SpareIn1 := 0.0, SpareIn2 := 0.0, CommonFirstOut := "CMN_FO", IsaAlarmFlashing := "UP".ALM_FLASHING, IsaTripFlashing := "UP".TRIP_FLASHING, Val_Out =>, Alm_Fail =>, Alm_HiHi =>, Alm_Hi =>, Alm_Lo =>, Alm_LoLo =>, Fo_Fail =>, Fo_HiHi =>, Fo_LoLo =>, SpareOut1 =>, SpareOut2 =>, SpareOut4 =>)
   END_RUNG
   // the same network as SCL:
   "LIT_33311"(Inp_PV := "LIT_33311_FLD",   // "SEID_AIn"
               Cfg_PVEUMin := "SETTINGS".LIT_33311.RANGE_L,
               Cfg_PVEUMax := "SETTINGS".LIT_33311.RANGE_H,
               Cfg_InpRawMin := 0,
               Cfg_InpRawMax := 27648,
               Cfg_FailRawHiLim := 29376,
               Cfg_FailRawLoLim := -691,
               Inp_PVBad := false,
               Cfg_FailBypass := false,
               Cfg_FailTripsUnit := true,
               Cfg_FailResetRequired := false,
               Cfg_InFailUsePVEUMax := "AlwaysTRUE",
               Cfg_InFailUsePVEUMin := "AlwaysFALSE",
               Cfg_InFailUseValSub := "AlwaysFALSE",
               Cfg_ValSub := 0.0,
               Cfg_FailDelay := T#0ms,
               Cfg_HasHiHiAlm := "AlwaysTRUE",
               Oset_HiHiLim := "SETTINGS".LIT_33311.SP_HH,
               Cfg_HiHiDelay := T#1s,
               Cfg_HiHiDB := 0.0,
               Cfg_HiHiBypass := false,
               Cfg_HiHiTripsUnit := true,
               Cfg_HiHiResetRequired := false,
               Cfg_HasHiAlm := "AlwaysTRUE",
               Oset_HiLim := "SETTINGS".LIT_33311.SP_H,
               Cfg_HiDelay := T#1s,
               Cfg_HiDB := 0.0,
               Cfg_HiBypass := false,
               Cfg_HiResetRequired := false,
               Cfg_HasLoAlm := "AlwaysFALSE",
               Oset_LoLim := "SETTINGS".LIT_33311.SP_L,
               Cfg_LoDelay := T#1s,
               Cfg_LoDB := 0.0,
               Cfg_LoBypass := false,
               Cfg_LoResetRequired := false,
               Cfg_HasLoLoAlm := "AlwaysFALSE",
               Oset_LoLoLim := "SETTINGS".LIT_33311.SP_LL,
               Cfg_LoLoDelay := T#1s,
               Cfg_LoLoDB := 0.0,
               Cfg_LoLoBypass := false,
               Cfg_LoLoTripsUnit := false,
               Cfg_LoLoResetRequired := false,
               Inp_Reset := "RESET",
               PCmd_MOS := false,
               SpareIn1 := 0.0,
               SpareIn2 := 0.0,
               CommonFirstOut := "CMN_FO",
               IsaAlarmFlashing := "UP".ALM_FLASHING,
               IsaTripFlashing := "UP".TRIP_FLASHING);
END_REGION

REGION Network 17: OIL PUMP A SEAL POT LEVEL
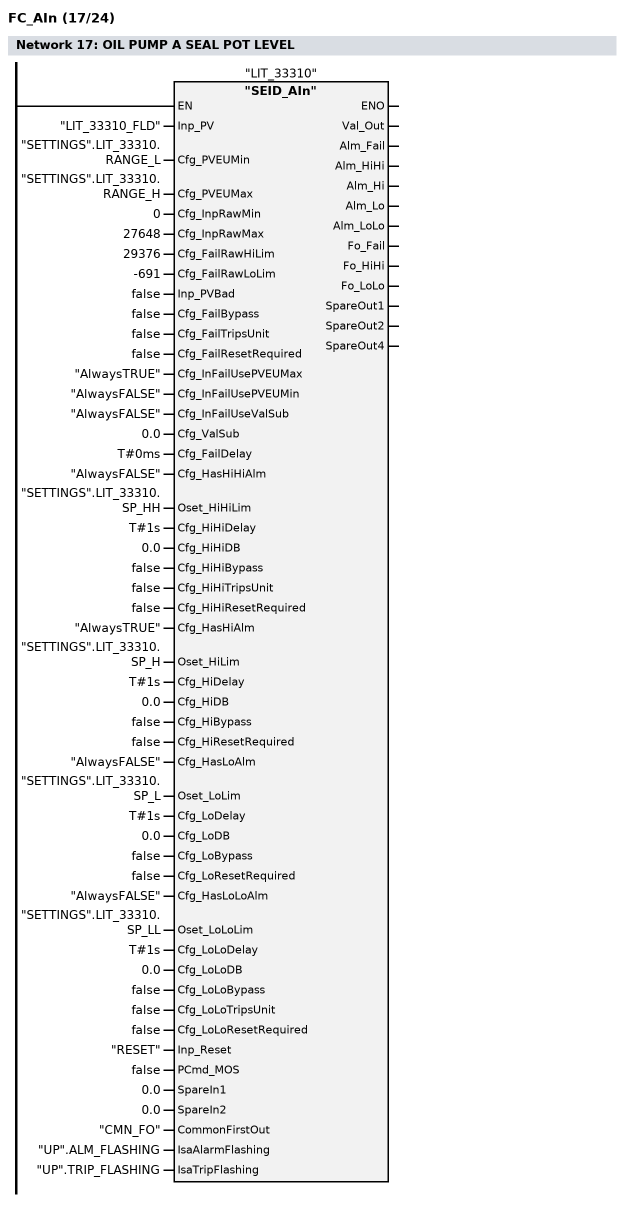
   RUNG wire#powerrail
      "LIT_33310"(Inp_PV := "LIT_33310_FLD", Cfg_PVEUMin := "SETTINGS".LIT_33310.RANGE_L, Cfg_PVEUMax := "SETTINGS".LIT_33310.RANGE_H, Cfg_InpRawMin := 0, Cfg_InpRawMax := 27648, Cfg_FailRawHiLim := 29376, Cfg_FailRawLoLim := -691, Inp_PVBad := false, Cfg_FailBypass := false, Cfg_FailTripsUnit := false, Cfg_FailResetRequired := false, Cfg_InFailUsePVEUMax := "AlwaysTRUE", Cfg_InFailUsePVEUMin := "AlwaysFALSE", Cfg_InFailUseValSub := "AlwaysFALSE", Cfg_ValSub := 0.0, Cfg_FailDelay := T#0ms, Cfg_HasHiHiAlm := "AlwaysFALSE", Oset_HiHiLim := "SETTINGS".LIT_33310.SP_HH, Cfg_HiHiDelay := T#1s, Cfg_HiHiDB := 0.0, Cfg_HiHiBypass := false, Cfg_HiHiTripsUnit := false, Cfg_HiHiResetRequired := false, Cfg_HasHiAlm := "AlwaysTRUE", Oset_HiLim := "SETTINGS".LIT_33310.SP_H, Cfg_HiDelay := T#1s, Cfg_HiDB := 0.0, Cfg_HiBypass := false, Cfg_HiResetRequired := false, Cfg_HasLoAlm := "AlwaysFALSE", Oset_LoLim := "SETTINGS".LIT_33310.SP_L, Cfg_LoDelay := T#1s, Cfg_LoDB := 0.0, Cfg_LoBypass := false, Cfg_LoResetRequired := false, Cfg_HasLoLoAlm := "AlwaysFALSE", Oset_LoLoLim := "SETTINGS".LIT_33310.SP_LL, Cfg_LoLoDelay := T#1s, Cfg_LoLoDB := 0.0, Cfg_LoLoBypass := false, Cfg_LoLoTripsUnit := false, Cfg_LoLoResetRequired := false, Inp_Reset := "RESET", PCmd_MOS := false, SpareIn1 := 0.0, SpareIn2 := 0.0, CommonFirstOut := "CMN_FO", IsaAlarmFlashing := "UP".ALM_FLASHING, IsaTripFlashing := "UP".TRIP_FLASHING, Val_Out =>, Alm_Fail =>, Alm_HiHi =>, Alm_Hi =>, Alm_Lo =>, Alm_LoLo =>, Fo_Fail =>, Fo_HiHi =>, Fo_LoLo =>, SpareOut1 =>, SpareOut2 =>, SpareOut4 =>)
   END_RUNG
   // the same network as SCL:
   "LIT_33310"(Inp_PV := "LIT_33310_FLD",   // "SEID_AIn"
               Cfg_PVEUMin := "SETTINGS".LIT_33310.RANGE_L,
               Cfg_PVEUMax := "SETTINGS".LIT_33310.RANGE_H,
               Cfg_InpRawMin := 0,
               Cfg_InpRawMax := 27648,
               Cfg_FailRawHiLim := 29376,
               Cfg_FailRawLoLim := -691,
               Inp_PVBad := false,
               Cfg_FailBypass := false,
               Cfg_FailTripsUnit := false,
               Cfg_FailResetRequired := false,
               Cfg_InFailUsePVEUMax := "AlwaysTRUE",
               Cfg_InFailUsePVEUMin := "AlwaysFALSE",
               Cfg_InFailUseValSub := "AlwaysFALSE",
               Cfg_ValSub := 0.0,
               Cfg_FailDelay := T#0ms,
               Cfg_HasHiHiAlm := "AlwaysFALSE",
               Oset_HiHiLim := "SETTINGS".LIT_33310.SP_HH,
               Cfg_HiHiDelay := T#1s,
               Cfg_HiHiDB := 0.0,
               Cfg_HiHiBypass := false,
               Cfg_HiHiTripsUnit := false,
               Cfg_HiHiResetRequired := false,
               Cfg_HasHiAlm := "AlwaysTRUE",
               Oset_HiLim := "SETTINGS".LIT_33310.SP_H,
               Cfg_HiDelay := T#1s,
               Cfg_HiDB := 0.0,
               Cfg_HiBypass := false,
               Cfg_HiResetRequired := false,
               Cfg_HasLoAlm := "AlwaysFALSE",
               Oset_LoLim := "SETTINGS".LIT_33310.SP_L,
               Cfg_LoDelay := T#1s,
               Cfg_LoDB := 0.0,
               Cfg_LoBypass := false,
               Cfg_LoResetRequired := false,
               Cfg_HasLoLoAlm := "AlwaysFALSE",
               Oset_LoLoLim := "SETTINGS".LIT_33310.SP_LL,
               Cfg_LoLoDelay := T#1s,
               Cfg_LoLoDB := 0.0,
               Cfg_LoLoBypass := false,
               Cfg_LoLoTripsUnit := false,
               Cfg_LoLoResetRequired := false,
               Inp_Reset := "RESET",
               PCmd_MOS := false,
               SpareIn1 := 0.0,
               SpareIn2 := 0.0,
               CommonFirstOut := "CMN_FO",
               IsaAlarmFlashing := "UP".ALM_FLASHING,
               IsaTripFlashing := "UP".TRIP_FLASHING);
END_REGION

REGION Network 18: OIL PUMP B SEAL POT LEVEL
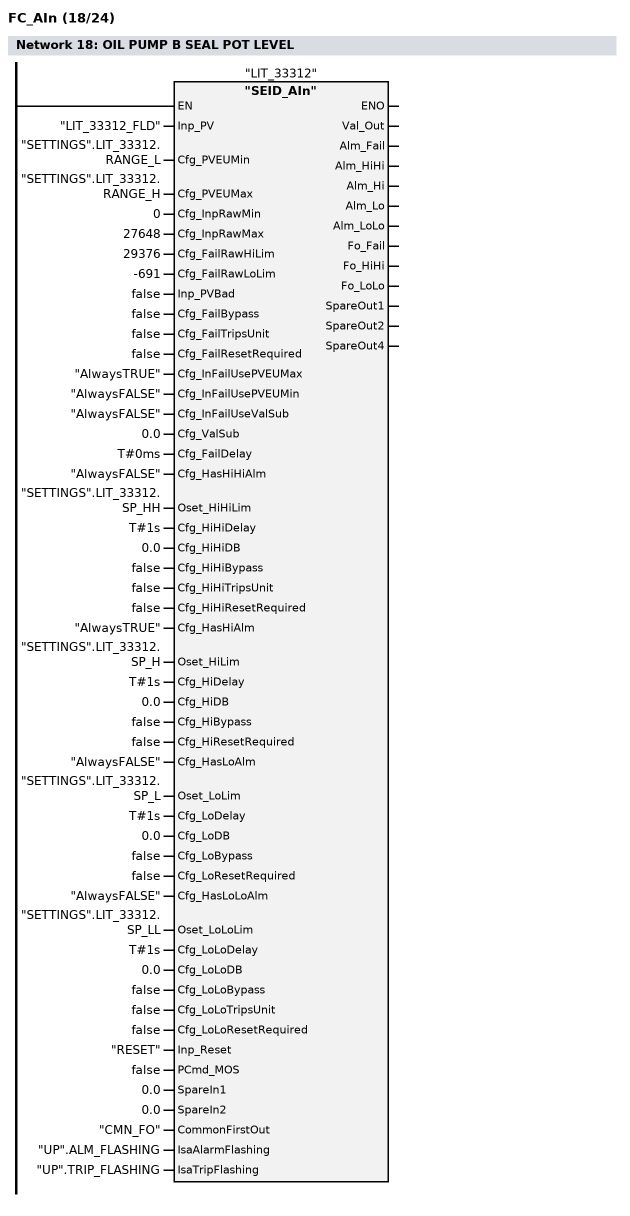
   RUNG wire#powerrail
      "LIT_33312"(Inp_PV := "LIT_33312_FLD", Cfg_PVEUMin := "SETTINGS".LIT_33312.RANGE_L, Cfg_PVEUMax := "SETTINGS".LIT_33312.RANGE_H, Cfg_InpRawMin := 0, Cfg_InpRawMax := 27648, Cfg_FailRawHiLim := 29376, Cfg_FailRawLoLim := -691, Inp_PVBad := false, Cfg_FailBypass := false, Cfg_FailTripsUnit := false, Cfg_FailResetRequired := false, Cfg_InFailUsePVEUMax := "AlwaysTRUE", Cfg_InFailUsePVEUMin := "AlwaysFALSE", Cfg_InFailUseValSub := "AlwaysFALSE", Cfg_ValSub := 0.0, Cfg_FailDelay := T#0ms, Cfg_HasHiHiAlm := "AlwaysFALSE", Oset_HiHiLim := "SETTINGS".LIT_33312.SP_HH, Cfg_HiHiDelay := T#1s, Cfg_HiHiDB := 0.0, Cfg_HiHiBypass := false, Cfg_HiHiTripsUnit := false, Cfg_HiHiResetRequired := false, Cfg_HasHiAlm := "AlwaysTRUE", Oset_HiLim := "SETTINGS".LIT_33312.SP_H, Cfg_HiDelay := T#1s, Cfg_HiDB := 0.0, Cfg_HiBypass := false, Cfg_HiResetRequired := false, Cfg_HasLoAlm := "AlwaysFALSE", Oset_LoLim := "SETTINGS".LIT_33312.SP_L, Cfg_LoDelay := T#1s, Cfg_LoDB := 0.0, Cfg_LoBypass := false, Cfg_LoResetRequired := false, Cfg_HasLoLoAlm := "AlwaysFALSE", Oset_LoLoLim := "SETTINGS".LIT_33312.SP_LL, Cfg_LoLoDelay := T#1s, Cfg_LoLoDB := 0.0, Cfg_LoLoBypass := false, Cfg_LoLoTripsUnit := false, Cfg_LoLoResetRequired := false, Inp_Reset := "RESET", PCmd_MOS := false, SpareIn1 := 0.0, SpareIn2 := 0.0, CommonFirstOut := "CMN_FO", IsaAlarmFlashing := "UP".ALM_FLASHING, IsaTripFlashing := "UP".TRIP_FLASHING, Val_Out =>, Alm_Fail =>, Alm_HiHi =>, Alm_Hi =>, Alm_Lo =>, Alm_LoLo =>, Fo_Fail =>, Fo_HiHi =>, Fo_LoLo =>, SpareOut1 =>, SpareOut2 =>, SpareOut4 =>)
   END_RUNG
   // the same network as SCL:
   "LIT_33312"(Inp_PV := "LIT_33312_FLD",   // "SEID_AIn"
               Cfg_PVEUMin := "SETTINGS".LIT_33312.RANGE_L,
               Cfg_PVEUMax := "SETTINGS".LIT_33312.RANGE_H,
               Cfg_InpRawMin := 0,
               Cfg_InpRawMax := 27648,
               Cfg_FailRawHiLim := 29376,
               Cfg_FailRawLoLim := -691,
               Inp_PVBad := false,
               Cfg_FailBypass := false,
               Cfg_FailTripsUnit := false,
               Cfg_FailResetRequired := false,
               Cfg_InFailUsePVEUMax := "AlwaysTRUE",
               Cfg_InFailUsePVEUMin := "AlwaysFALSE",
               Cfg_InFailUseValSub := "AlwaysFALSE",
               Cfg_ValSub := 0.0,
               Cfg_FailDelay := T#0ms,
               Cfg_HasHiHiAlm := "AlwaysFALSE",
               Oset_HiHiLim := "SETTINGS".LIT_33312.SP_HH,
               Cfg_HiHiDelay := T#1s,
               Cfg_HiHiDB := 0.0,
               Cfg_HiHiBypass := false,
               Cfg_HiHiTripsUnit := false,
               Cfg_HiHiResetRequired := false,
               Cfg_HasHiAlm := "AlwaysTRUE",
               Oset_HiLim := "SETTINGS".LIT_33312.SP_H,
               Cfg_HiDelay := T#1s,
               Cfg_HiDB := 0.0,
               Cfg_HiBypass := false,
               Cfg_HiResetRequired := false,
               Cfg_HasLoAlm := "AlwaysFALSE",
               Oset_LoLim := "SETTINGS".LIT_33312.SP_L,
               Cfg_LoDelay := T#1s,
               Cfg_LoDB := 0.0,
               Cfg_LoBypass := false,
               Cfg_LoResetRequired := false,
               Cfg_HasLoLoAlm := "AlwaysFALSE",
               Oset_LoLoLim := "SETTINGS".LIT_33312.SP_LL,
               Cfg_LoLoDelay := T#1s,
               Cfg_LoLoDB := 0.0,
               Cfg_LoLoBypass := false,
               Cfg_LoLoTripsUnit := false,
               Cfg_LoLoResetRequired := false,
               Inp_Reset := "RESET",
               PCmd_MOS := false,
               SpareIn1 := 0.0,
               SpareIn2 := 0.0,
               CommonFirstOut := "CMN_FO",
               IsaAlarmFlashing := "UP".ALM_FLASHING,
               IsaTripFlashing := "UP".TRIP_FLASHING);
END_REGION

REGION Network 19: OIL PUMP A SEAL POT PRESSURE
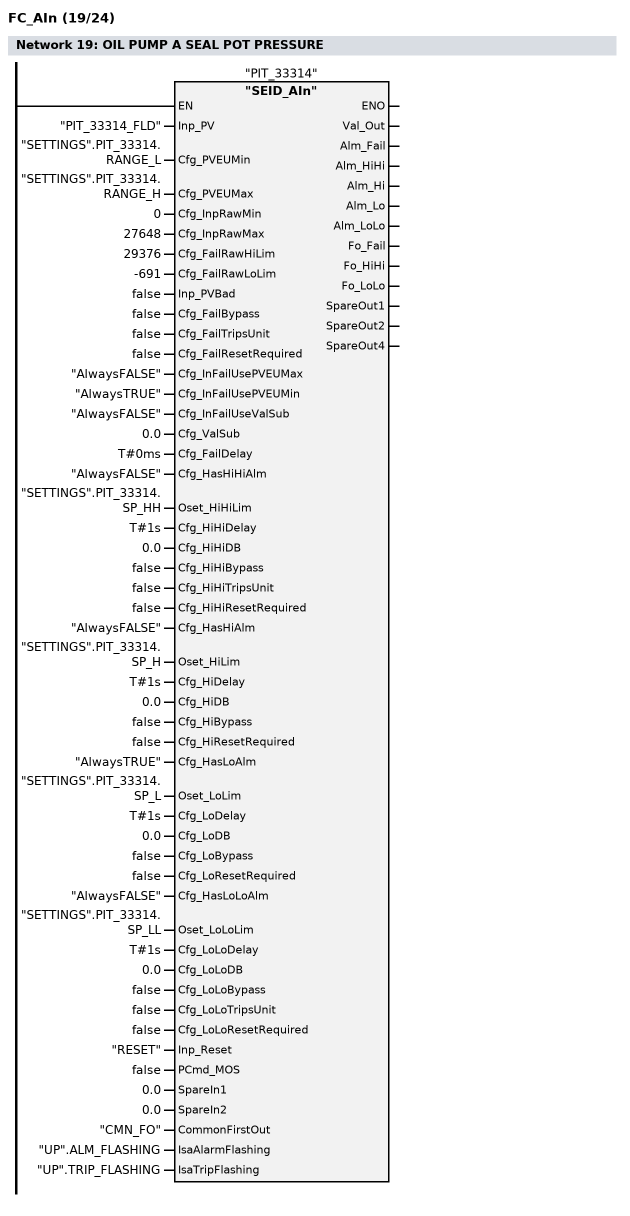
   RUNG wire#powerrail
      "PIT_33314"(Inp_PV := "PIT_33314_FLD", Cfg_PVEUMin := "SETTINGS".PIT_33314.RANGE_L, Cfg_PVEUMax := "SETTINGS".PIT_33314.RANGE_H, Cfg_InpRawMin := 0, Cfg_InpRawMax := 27648, Cfg_FailRawHiLim := 29376, Cfg_FailRawLoLim := -691, Inp_PVBad := false, Cfg_FailBypass := false, Cfg_FailTripsUnit := false, Cfg_FailResetRequired := false, Cfg_InFailUsePVEUMax := "AlwaysFALSE", Cfg_InFailUsePVEUMin := "AlwaysTRUE", Cfg_InFailUseValSub := "AlwaysFALSE", Cfg_ValSub := 0.0, Cfg_FailDelay := T#0ms, Cfg_HasHiHiAlm := "AlwaysFALSE", Oset_HiHiLim := "SETTINGS".PIT_33314.SP_HH, Cfg_HiHiDelay := T#1s, Cfg_HiHiDB := 0.0, Cfg_HiHiBypass := false, Cfg_HiHiTripsUnit := false, Cfg_HiHiResetRequired := false, Cfg_HasHiAlm := "AlwaysFALSE", Oset_HiLim := "SETTINGS".PIT_33314.SP_H, Cfg_HiDelay := T#1s, Cfg_HiDB := 0.0, Cfg_HiBypass := false, Cfg_HiResetRequired := false, Cfg_HasLoAlm := "AlwaysTRUE", Oset_LoLim := "SETTINGS".PIT_33314.SP_L, Cfg_LoDelay := T#1s, Cfg_LoDB := 0.0, Cfg_LoBypass := false, Cfg_LoResetRequired := false, Cfg_HasLoLoAlm := "AlwaysFALSE", Oset_LoLoLim := "SETTINGS".PIT_33314.SP_LL, Cfg_LoLoDelay := T#1s, Cfg_LoLoDB := 0.0, Cfg_LoLoBypass := false, Cfg_LoLoTripsUnit := false, Cfg_LoLoResetRequired := false, Inp_Reset := "RESET", PCmd_MOS := false, SpareIn1 := 0.0, SpareIn2 := 0.0, CommonFirstOut := "CMN_FO", IsaAlarmFlashing := "UP".ALM_FLASHING, IsaTripFlashing := "UP".TRIP_FLASHING, Val_Out =>, Alm_Fail =>, Alm_HiHi =>, Alm_Hi =>, Alm_Lo =>, Alm_LoLo =>, Fo_Fail =>, Fo_HiHi =>, Fo_LoLo =>, SpareOut1 =>, SpareOut2 =>, SpareOut4 =>)
   END_RUNG
   // the same network as SCL:
   "PIT_33314"(Inp_PV := "PIT_33314_FLD",   // "SEID_AIn"
               Cfg_PVEUMin := "SETTINGS".PIT_33314.RANGE_L,
               Cfg_PVEUMax := "SETTINGS".PIT_33314.RANGE_H,
               Cfg_InpRawMin := 0,
               Cfg_InpRawMax := 27648,
               Cfg_FailRawHiLim := 29376,
               Cfg_FailRawLoLim := -691,
               Inp_PVBad := false,
               Cfg_FailBypass := false,
               Cfg_FailTripsUnit := false,
               Cfg_FailResetRequired := false,
               Cfg_InFailUsePVEUMax := "AlwaysFALSE",
               Cfg_InFailUsePVEUMin := "AlwaysTRUE",
               Cfg_InFailUseValSub := "AlwaysFALSE",
               Cfg_ValSub := 0.0,
               Cfg_FailDelay := T#0ms,
               Cfg_HasHiHiAlm := "AlwaysFALSE",
               Oset_HiHiLim := "SETTINGS".PIT_33314.SP_HH,
               Cfg_HiHiDelay := T#1s,
               Cfg_HiHiDB := 0.0,
               Cfg_HiHiBypass := false,
               Cfg_HiHiTripsUnit := false,
               Cfg_HiHiResetRequired := false,
               Cfg_HasHiAlm := "AlwaysFALSE",
               Oset_HiLim := "SETTINGS".PIT_33314.SP_H,
               Cfg_HiDelay := T#1s,
               Cfg_HiDB := 0.0,
               Cfg_HiBypass := false,
               Cfg_HiResetRequired := false,
               Cfg_HasLoAlm := "AlwaysTRUE",
               Oset_LoLim := "SETTINGS".PIT_33314.SP_L,
               Cfg_LoDelay := T#1s,
               Cfg_LoDB := 0.0,
               Cfg_LoBypass := false,
               Cfg_LoResetRequired := false,
               Cfg_HasLoLoAlm := "AlwaysFALSE",
               Oset_LoLoLim := "SETTINGS".PIT_33314.SP_LL,
               Cfg_LoLoDelay := T#1s,
               Cfg_LoLoDB := 0.0,
               Cfg_LoLoBypass := false,
               Cfg_LoLoTripsUnit := false,
               Cfg_LoLoResetRequired := false,
               Inp_Reset := "RESET",
               PCmd_MOS := false,
               SpareIn1 := 0.0,
               SpareIn2 := 0.0,
               CommonFirstOut := "CMN_FO",
               IsaAlarmFlashing := "UP".ALM_FLASHING,
               IsaTripFlashing := "UP".TRIP_FLASHING);
END_REGION

REGION Network 20: OIL PUMP B SEAL POT PRESSURE
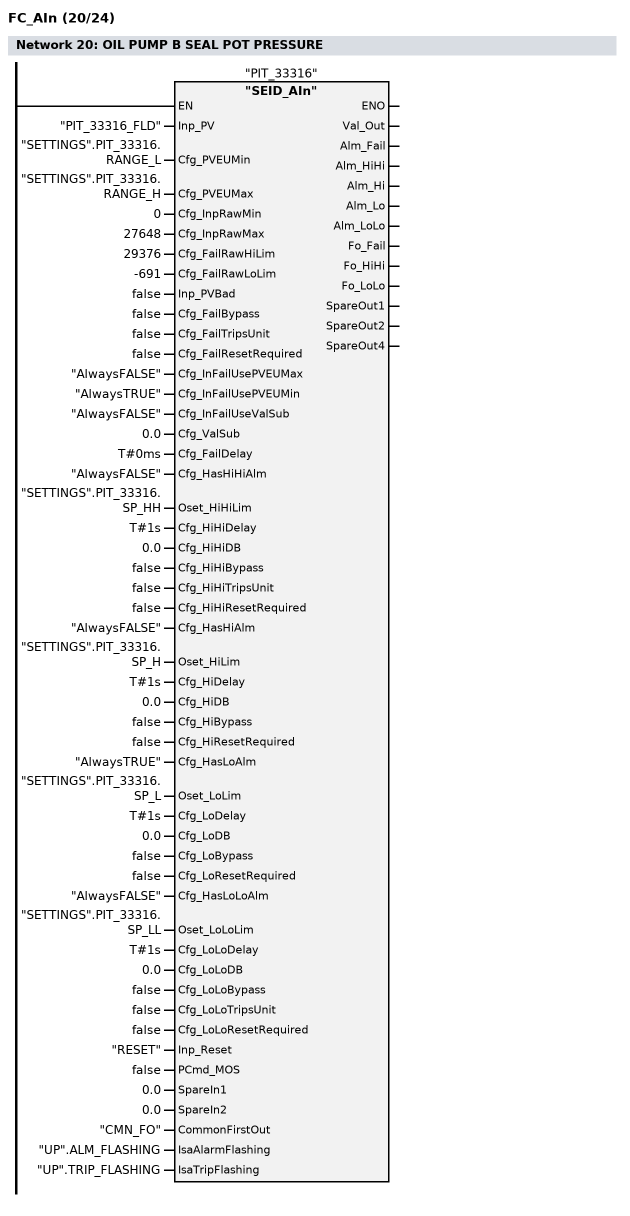
   RUNG wire#powerrail
      "PIT_33316"(Inp_PV := "PIT_33316_FLD", Cfg_PVEUMin := "SETTINGS".PIT_33316.RANGE_L, Cfg_PVEUMax := "SETTINGS".PIT_33316.RANGE_H, Cfg_InpRawMin := 0, Cfg_InpRawMax := 27648, Cfg_FailRawHiLim := 29376, Cfg_FailRawLoLim := -691, Inp_PVBad := false, Cfg_FailBypass := false, Cfg_FailTripsUnit := false, Cfg_FailResetRequired := false, Cfg_InFailUsePVEUMax := "AlwaysFALSE", Cfg_InFailUsePVEUMin := "AlwaysTRUE", Cfg_InFailUseValSub := "AlwaysFALSE", Cfg_ValSub := 0.0, Cfg_FailDelay := T#0ms, Cfg_HasHiHiAlm := "AlwaysFALSE", Oset_HiHiLim := "SETTINGS".PIT_33316.SP_HH, Cfg_HiHiDelay := T#1s, Cfg_HiHiDB := 0.0, Cfg_HiHiBypass := false, Cfg_HiHiTripsUnit := false, Cfg_HiHiResetRequired := false, Cfg_HasHiAlm := "AlwaysFALSE", Oset_HiLim := "SETTINGS".PIT_33316.SP_H, Cfg_HiDelay := T#1s, Cfg_HiDB := 0.0, Cfg_HiBypass := false, Cfg_HiResetRequired := false, Cfg_HasLoAlm := "AlwaysTRUE", Oset_LoLim := "SETTINGS".PIT_33316.SP_L, Cfg_LoDelay := T#1s, Cfg_LoDB := 0.0, Cfg_LoBypass := false, Cfg_LoResetRequired := false, Cfg_HasLoLoAlm := "AlwaysFALSE", Oset_LoLoLim := "SETTINGS".PIT_33316.SP_LL, Cfg_LoLoDelay := T#1s, Cfg_LoLoDB := 0.0, Cfg_LoLoBypass := false, Cfg_LoLoTripsUnit := false, Cfg_LoLoResetRequired := false, Inp_Reset := "RESET", PCmd_MOS := false, SpareIn1 := 0.0, SpareIn2 := 0.0, CommonFirstOut := "CMN_FO", IsaAlarmFlashing := "UP".ALM_FLASHING, IsaTripFlashing := "UP".TRIP_FLASHING, Val_Out =>, Alm_Fail =>, Alm_HiHi =>, Alm_Hi =>, Alm_Lo =>, Alm_LoLo =>, Fo_Fail =>, Fo_HiHi =>, Fo_LoLo =>, SpareOut1 =>, SpareOut2 =>, SpareOut4 =>)
   END_RUNG
   // the same network as SCL:
   "PIT_33316"(Inp_PV := "PIT_33316_FLD",   // "SEID_AIn"
               Cfg_PVEUMin := "SETTINGS".PIT_33316.RANGE_L,
               Cfg_PVEUMax := "SETTINGS".PIT_33316.RANGE_H,
               Cfg_InpRawMin := 0,
               Cfg_InpRawMax := 27648,
               Cfg_FailRawHiLim := 29376,
               Cfg_FailRawLoLim := -691,
               Inp_PVBad := false,
               Cfg_FailBypass := false,
               Cfg_FailTripsUnit := false,
               Cfg_FailResetRequired := false,
               Cfg_InFailUsePVEUMax := "AlwaysFALSE",
               Cfg_InFailUsePVEUMin := "AlwaysTRUE",
               Cfg_InFailUseValSub := "AlwaysFALSE",
               Cfg_ValSub := 0.0,
               Cfg_FailDelay := T#0ms,
               Cfg_HasHiHiAlm := "AlwaysFALSE",
               Oset_HiHiLim := "SETTINGS".PIT_33316.SP_HH,
               Cfg_HiHiDelay := T#1s,
               Cfg_HiHiDB := 0.0,
               Cfg_HiHiBypass := false,
               Cfg_HiHiTripsUnit := false,
               Cfg_HiHiResetRequired := false,
               Cfg_HasHiAlm := "AlwaysFALSE",
               Oset_HiLim := "SETTINGS".PIT_33316.SP_H,
               Cfg_HiDelay := T#1s,
               Cfg_HiDB := 0.0,
               Cfg_HiBypass := false,
               Cfg_HiResetRequired := false,
               Cfg_HasLoAlm := "AlwaysTRUE",
               Oset_LoLim := "SETTINGS".PIT_33316.SP_L,
               Cfg_LoDelay := T#1s,
               Cfg_LoDB := 0.0,
               Cfg_LoBypass := false,
               Cfg_LoResetRequired := false,
               Cfg_HasLoLoAlm := "AlwaysFALSE",
               Oset_LoLoLim := "SETTINGS".PIT_33316.SP_LL,
               Cfg_LoLoDelay := T#1s,
               Cfg_LoLoDB := 0.0,
               Cfg_LoLoBypass := false,
               Cfg_LoLoTripsUnit := false,
               Cfg_LoLoResetRequired := false,
               Inp_Reset := "RESET",
               PCmd_MOS := false,
               SpareIn1 := 0.0,
               SpareIn2 := 0.0,
               CommonFirstOut := "CMN_FO",
               IsaAlarmFlashing := "UP".ALM_FLASHING,
               IsaTripFlashing := "UP".TRIP_FLASHING);
END_REGION

REGION Network 21: OIL SEPARATOR TEMPERATURE
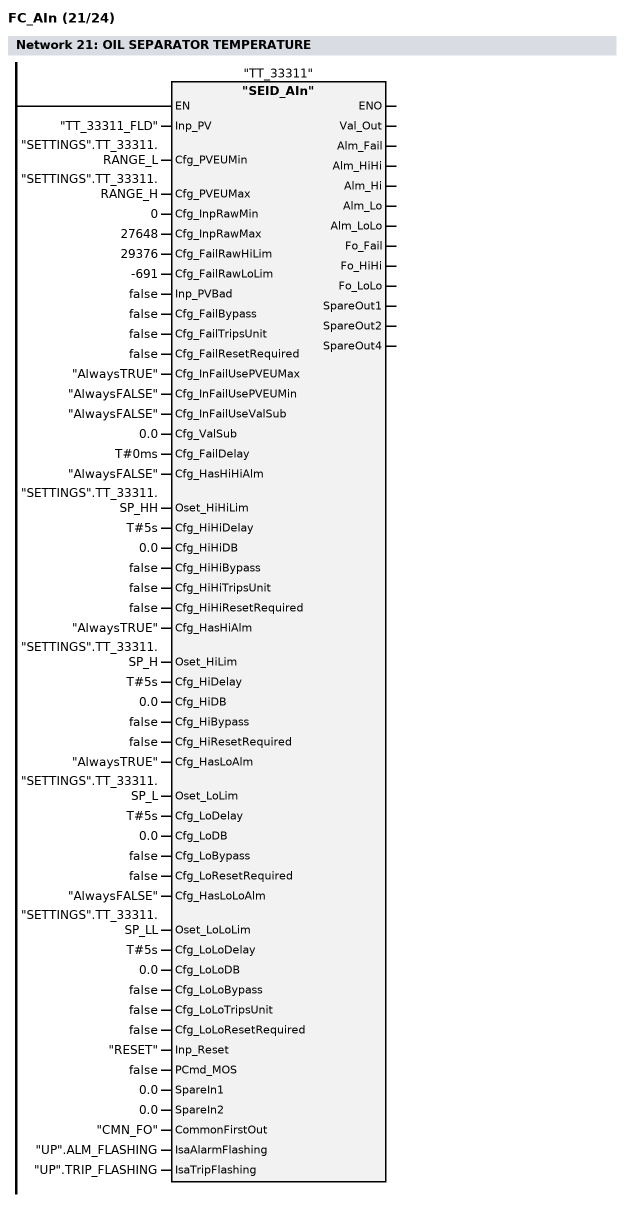
   RUNG wire#powerrail
      "TT_33311"(Inp_PV := "TT_33311_FLD", Cfg_PVEUMin := "SETTINGS".TT_33311.RANGE_L, Cfg_PVEUMax := "SETTINGS".TT_33311.RANGE_H, Cfg_InpRawMin := 0, Cfg_InpRawMax := 27648, Cfg_FailRawHiLim := 29376, Cfg_FailRawLoLim := -691, Inp_PVBad := false, Cfg_FailBypass := false, Cfg_FailTripsUnit := false, Cfg_FailResetRequired := false, Cfg_InFailUsePVEUMax := "AlwaysTRUE", Cfg_InFailUsePVEUMin := "AlwaysFALSE", Cfg_InFailUseValSub := "AlwaysFALSE", Cfg_ValSub := 0.0, Cfg_FailDelay := T#0ms, Cfg_HasHiHiAlm := "AlwaysFALSE", Oset_HiHiLim := "SETTINGS".TT_33311.SP_HH, Cfg_HiHiDelay := T#5s, Cfg_HiHiDB := 0.0, Cfg_HiHiBypass := false, Cfg_HiHiTripsUnit := false, Cfg_HiHiResetRequired := false, Cfg_HasHiAlm := "AlwaysTRUE", Oset_HiLim := "SETTINGS".TT_33311.SP_H, Cfg_HiDelay := T#5s, Cfg_HiDB := 0.0, Cfg_HiBypass := false, Cfg_HiResetRequired := false, Cfg_HasLoAlm := "AlwaysTRUE", Oset_LoLim := "SETTINGS".TT_33311.SP_L, Cfg_LoDelay := T#5s, Cfg_LoDB := 0.0, Cfg_LoBypass := false, Cfg_LoResetRequired := false, Cfg_HasLoLoAlm := "AlwaysFALSE", Oset_LoLoLim := "SETTINGS".TT_33311.SP_LL, Cfg_LoLoDelay := T#5s, Cfg_LoLoDB := 0.0, Cfg_LoLoBypass := false, Cfg_LoLoTripsUnit := false, Cfg_LoLoResetRequired := false, Inp_Reset := "RESET", PCmd_MOS := false, SpareIn1 := 0.0, SpareIn2 := 0.0, CommonFirstOut := "CMN_FO", IsaAlarmFlashing := "UP".ALM_FLASHING, IsaTripFlashing := "UP".TRIP_FLASHING, Val_Out =>, Alm_Fail =>, Alm_HiHi =>, Alm_Hi =>, Alm_Lo =>, Alm_LoLo =>, Fo_Fail =>, Fo_HiHi =>, Fo_LoLo =>, SpareOut1 =>, SpareOut2 =>, SpareOut4 =>)
   END_RUNG
   // the same network as SCL:
   "TT_33311"(Inp_PV := "TT_33311_FLD",   // "SEID_AIn"
              Cfg_PVEUMin := "SETTINGS".TT_33311.RANGE_L,
              Cfg_PVEUMax := "SETTINGS".TT_33311.RANGE_H,
              Cfg_InpRawMin := 0,
              Cfg_InpRawMax := 27648,
              Cfg_FailRawHiLim := 29376,
              Cfg_FailRawLoLim := -691,
              Inp_PVBad := false,
              Cfg_FailBypass := false,
              Cfg_FailTripsUnit := false,
              Cfg_FailResetRequired := false,
              Cfg_InFailUsePVEUMax := "AlwaysTRUE",
              Cfg_InFailUsePVEUMin := "AlwaysFALSE",
              Cfg_InFailUseValSub := "AlwaysFALSE",
              Cfg_ValSub := 0.0,
              Cfg_FailDelay := T#0ms,
              Cfg_HasHiHiAlm := "AlwaysFALSE",
              Oset_HiHiLim := "SETTINGS".TT_33311.SP_HH,
              Cfg_HiHiDelay := T#5s,
              Cfg_HiHiDB := 0.0,
              Cfg_HiHiBypass := false,
              Cfg_HiHiTripsUnit := false,
              Cfg_HiHiResetRequired := false,
              Cfg_HasHiAlm := "AlwaysTRUE",
              Oset_HiLim := "SETTINGS".TT_33311.SP_H,
              Cfg_HiDelay := T#5s,
              Cfg_HiDB := 0.0,
              Cfg_HiBypass := false,
              Cfg_HiResetRequired := false,
              Cfg_HasLoAlm := "AlwaysTRUE",
              Oset_LoLim := "SETTINGS".TT_33311.SP_L,
              Cfg_LoDelay := T#5s,
              Cfg_LoDB := 0.0,
              Cfg_LoBypass := false,
              Cfg_LoResetRequired := false,
              Cfg_HasLoLoAlm := "AlwaysFALSE",
              Oset_LoLoLim := "SETTINGS".TT_33311.SP_LL,
              Cfg_LoLoDelay := T#5s,
              Cfg_LoLoDB := 0.0,
              Cfg_LoLoBypass := false,
              Cfg_LoLoTripsUnit := false,
              Cfg_LoLoResetRequired := false,
              Inp_Reset := "RESET",
              PCmd_MOS := false,
              SpareIn1 := 0.0,
              SpareIn2 := 0.0,
              CommonFirstOut := "CMN_FO",
              IsaAlarmFlashing := "UP".ALM_FLASHING,
              IsaTripFlashing := "UP".TRIP_FLASHING);
END_REGION

REGION Network 22: COMPRESSOR SEAL POT PRESSURE
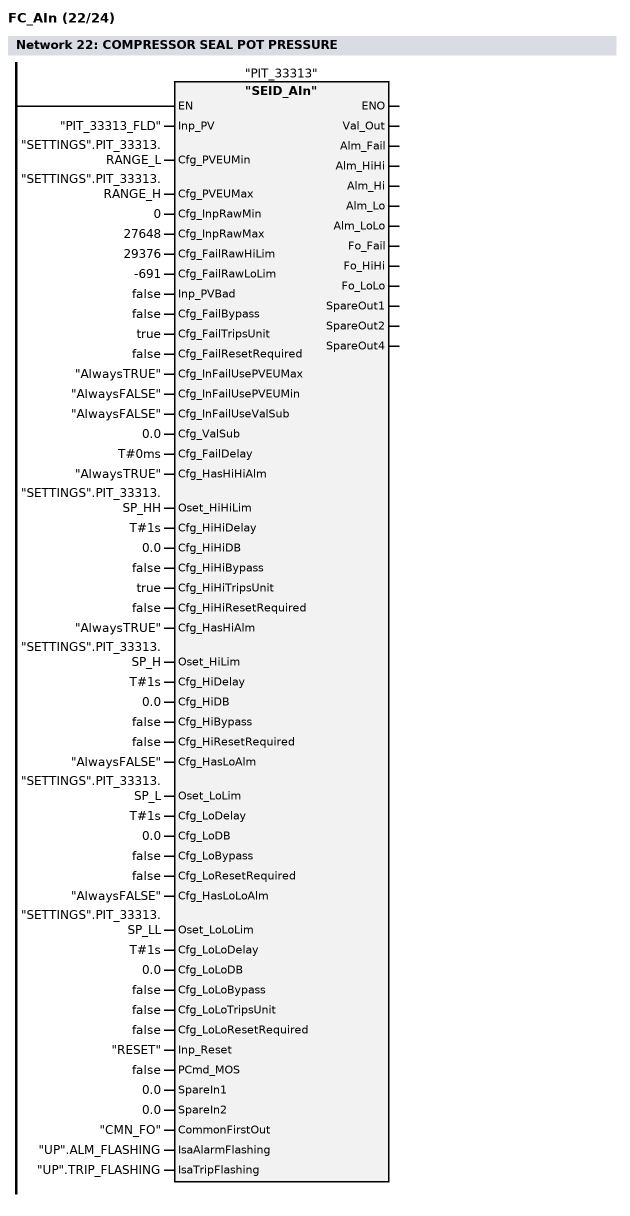
   RUNG wire#powerrail
      "PIT_33313"(Inp_PV := "PIT_33313_FLD", Cfg_PVEUMin := "SETTINGS".PIT_33313.RANGE_L, Cfg_PVEUMax := "SETTINGS".PIT_33313.RANGE_H, Cfg_InpRawMin := 0, Cfg_InpRawMax := 27648, Cfg_FailRawHiLim := 29376, Cfg_FailRawLoLim := -691, Inp_PVBad := false, Cfg_FailBypass := false, Cfg_FailTripsUnit := true, Cfg_FailResetRequired := false, Cfg_InFailUsePVEUMax := "AlwaysTRUE", Cfg_InFailUsePVEUMin := "AlwaysFALSE", Cfg_InFailUseValSub := "AlwaysFALSE", Cfg_ValSub := 0.0, Cfg_FailDelay := T#0ms, Cfg_HasHiHiAlm := "AlwaysTRUE", Oset_HiHiLim := "SETTINGS".PIT_33313.SP_HH, Cfg_HiHiDelay := T#1s, Cfg_HiHiDB := 0.0, Cfg_HiHiBypass := false, Cfg_HiHiTripsUnit := true, Cfg_HiHiResetRequired := false, Cfg_HasHiAlm := "AlwaysTRUE", Oset_HiLim := "SETTINGS".PIT_33313.SP_H, Cfg_HiDelay := T#1s, Cfg_HiDB := 0.0, Cfg_HiBypass := false, Cfg_HiResetRequired := false, Cfg_HasLoAlm := "AlwaysFALSE", Oset_LoLim := "SETTINGS".PIT_33313.SP_L, Cfg_LoDelay := T#1s, Cfg_LoDB := 0.0, Cfg_LoBypass := false, Cfg_LoResetRequired := false, Cfg_HasLoLoAlm := "AlwaysFALSE", Oset_LoLoLim := "SETTINGS".PIT_33313.SP_LL, Cfg_LoLoDelay := T#1s, Cfg_LoLoDB := 0.0, Cfg_LoLoBypass := false, Cfg_LoLoTripsUnit := false, Cfg_LoLoResetRequired := false, Inp_Reset := "RESET", PCmd_MOS := false, SpareIn1 := 0.0, SpareIn2 := 0.0, CommonFirstOut := "CMN_FO", IsaAlarmFlashing := "UP".ALM_FLASHING, IsaTripFlashing := "UP".TRIP_FLASHING, Val_Out =>, Alm_Fail =>, Alm_HiHi =>, Alm_Hi =>, Alm_Lo =>, Alm_LoLo =>, Fo_Fail =>, Fo_HiHi =>, Fo_LoLo =>, SpareOut1 =>, SpareOut2 =>, SpareOut4 =>)
   END_RUNG
   // the same network as SCL:
   "PIT_33313"(Inp_PV := "PIT_33313_FLD",   // "SEID_AIn"
               Cfg_PVEUMin := "SETTINGS".PIT_33313.RANGE_L,
               Cfg_PVEUMax := "SETTINGS".PIT_33313.RANGE_H,
               Cfg_InpRawMin := 0,
               Cfg_InpRawMax := 27648,
               Cfg_FailRawHiLim := 29376,
               Cfg_FailRawLoLim := -691,
               Inp_PVBad := false,
               Cfg_FailBypass := false,
               Cfg_FailTripsUnit := true,
               Cfg_FailResetRequired := false,
               Cfg_InFailUsePVEUMax := "AlwaysTRUE",
               Cfg_InFailUsePVEUMin := "AlwaysFALSE",
               Cfg_InFailUseValSub := "AlwaysFALSE",
               Cfg_ValSub := 0.0,
               Cfg_FailDelay := T#0ms,
               Cfg_HasHiHiAlm := "AlwaysTRUE",
               Oset_HiHiLim := "SETTINGS".PIT_33313.SP_HH,
               Cfg_HiHiDelay := T#1s,
               Cfg_HiHiDB := 0.0,
               Cfg_HiHiBypass := false,
               Cfg_HiHiTripsUnit := true,
               Cfg_HiHiResetRequired := false,
               Cfg_HasHiAlm := "AlwaysTRUE",
               Oset_HiLim := "SETTINGS".PIT_33313.SP_H,
               Cfg_HiDelay := T#1s,
               Cfg_HiDB := 0.0,
               Cfg_HiBypass := false,
               Cfg_HiResetRequired := false,
               Cfg_HasLoAlm := "AlwaysFALSE",
               Oset_LoLim := "SETTINGS".PIT_33313.SP_L,
               Cfg_LoDelay := T#1s,
               Cfg_LoDB := 0.0,
               Cfg_LoBypass := false,
               Cfg_LoResetRequired := false,
               Cfg_HasLoLoAlm := "AlwaysFALSE",
               Oset_LoLoLim := "SETTINGS".PIT_33313.SP_LL,
               Cfg_LoLoDelay := T#1s,
               Cfg_LoLoDB := 0.0,
               Cfg_LoLoBypass := false,
               Cfg_LoLoTripsUnit := false,
               Cfg_LoLoResetRequired := false,
               Inp_Reset := "RESET",
               PCmd_MOS := false,
               SpareIn1 := 0.0,
               SpareIn2 := 0.0,
               CommonFirstOut := "CMN_FO",
               IsaAlarmFlashing := "UP".ALM_FLASHING,
               IsaTripFlashing := "UP".TRIP_FLASHING);
END_REGION

REGION Network 23: COMPRESSOR MAIN MOTOR CURRENT
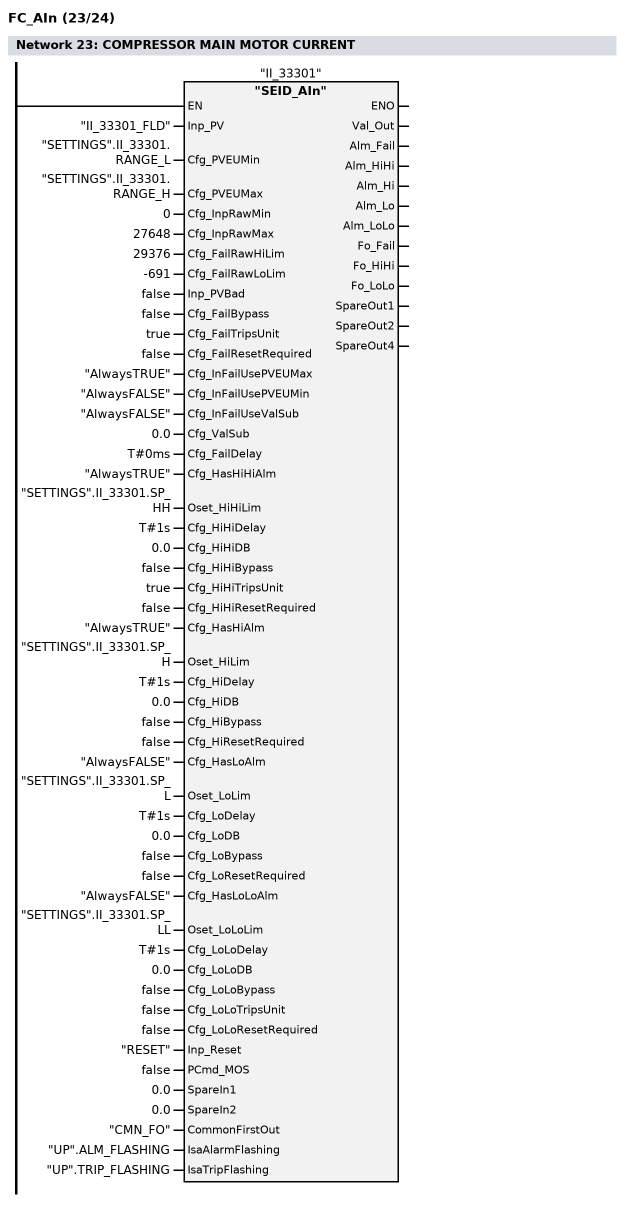
   RUNG wire#powerrail
      "II_33301"(Inp_PV := "II_33301_FLD", Cfg_PVEUMin := "SETTINGS".II_33301.RANGE_L, Cfg_PVEUMax := "SETTINGS".II_33301.RANGE_H, Cfg_InpRawMin := 0, Cfg_InpRawMax := 27648, Cfg_FailRawHiLim := 29376, Cfg_FailRawLoLim := -691, Inp_PVBad := false, Cfg_FailBypass := false, Cfg_FailTripsUnit := true, Cfg_FailResetRequired := false, Cfg_InFailUsePVEUMax := "AlwaysTRUE", Cfg_InFailUsePVEUMin := "AlwaysFALSE", Cfg_InFailUseValSub := "AlwaysFALSE", Cfg_ValSub := 0.0, Cfg_FailDelay := T#0ms, Cfg_HasHiHiAlm := "AlwaysTRUE", Oset_HiHiLim := "SETTINGS".II_33301.SP_HH, Cfg_HiHiDelay := T#1s, Cfg_HiHiDB := 0.0, Cfg_HiHiBypass := false, Cfg_HiHiTripsUnit := true, Cfg_HiHiResetRequired := false, Cfg_HasHiAlm := "AlwaysTRUE", Oset_HiLim := "SETTINGS".II_33301.SP_H, Cfg_HiDelay := T#1s, Cfg_HiDB := 0.0, Cfg_HiBypass := false, Cfg_HiResetRequired := false, Cfg_HasLoAlm := "AlwaysFALSE", Oset_LoLim := "SETTINGS".II_33301.SP_L, Cfg_LoDelay := T#1s, Cfg_LoDB := 0.0, Cfg_LoBypass := false, Cfg_LoResetRequired := false, Cfg_HasLoLoAlm := "AlwaysFALSE", Oset_LoLoLim := "SETTINGS".II_33301.SP_LL, Cfg_LoLoDelay := T#1s, Cfg_LoLoDB := 0.0, Cfg_LoLoBypass := false, Cfg_LoLoTripsUnit := false, Cfg_LoLoResetRequired := false, Inp_Reset := "RESET", PCmd_MOS := false, SpareIn1 := 0.0, SpareIn2 := 0.0, CommonFirstOut := "CMN_FO", IsaAlarmFlashing := "UP".ALM_FLASHING, IsaTripFlashing := "UP".TRIP_FLASHING, Val_Out =>, Alm_Fail =>, Alm_HiHi =>, Alm_Hi =>, Alm_Lo =>, Alm_LoLo =>, Fo_Fail =>, Fo_HiHi =>, Fo_LoLo =>, SpareOut1 =>, SpareOut2 =>, SpareOut4 =>)
   END_RUNG
   // the same network as SCL:
   "II_33301"(Inp_PV := "II_33301_FLD",   // "SEID_AIn"
              Cfg_PVEUMin := "SETTINGS".II_33301.RANGE_L,
              Cfg_PVEUMax := "SETTINGS".II_33301.RANGE_H,
              Cfg_InpRawMin := 0,
              Cfg_InpRawMax := 27648,
              Cfg_FailRawHiLim := 29376,
              Cfg_FailRawLoLim := -691,
              Inp_PVBad := false,
              Cfg_FailBypass := false,
              Cfg_FailTripsUnit := true,
              Cfg_FailResetRequired := false,
              Cfg_InFailUsePVEUMax := "AlwaysTRUE",
              Cfg_InFailUsePVEUMin := "AlwaysFALSE",
              Cfg_InFailUseValSub := "AlwaysFALSE",
              Cfg_ValSub := 0.0,
              Cfg_FailDelay := T#0ms,
              Cfg_HasHiHiAlm := "AlwaysTRUE",
              Oset_HiHiLim := "SETTINGS".II_33301.SP_HH,
              Cfg_HiHiDelay := T#1s,
              Cfg_HiHiDB := 0.0,
              Cfg_HiHiBypass := false,
              Cfg_HiHiTripsUnit := true,
              Cfg_HiHiResetRequired := false,
              Cfg_HasHiAlm := "AlwaysTRUE",
              Oset_HiLim := "SETTINGS".II_33301.SP_H,
              Cfg_HiDelay := T#1s,
              Cfg_HiDB := 0.0,
              Cfg_HiBypass := false,
              Cfg_HiResetRequired := false,
              Cfg_HasLoAlm := "AlwaysFALSE",
              Oset_LoLim := "SETTINGS".II_33301.SP_L,
              Cfg_LoDelay := T#1s,
              Cfg_LoDB := 0.0,
              Cfg_LoBypass := false,
              Cfg_LoResetRequired := false,
              Cfg_HasLoLoAlm := "AlwaysFALSE",
              Oset_LoLoLim := "SETTINGS".II_33301.SP_LL,
              Cfg_LoLoDelay := T#1s,
              Cfg_LoLoDB := 0.0,
              Cfg_LoLoBypass := false,
              Cfg_LoLoTripsUnit := false,
              Cfg_LoLoResetRequired := false,
              Inp_Reset := "RESET",
              PCmd_MOS := false,
              SpareIn1 := 0.0,
              SpareIn2 := 0.0,
              CommonFirstOut := "CMN_FO",
              IsaAlarmFlashing := "UP".ALM_FLASHING,
              IsaTripFlashing := "UP".TRIP_FLASHING);
END_REGION

REGION Network 24: SLIDE VALVE POSITION
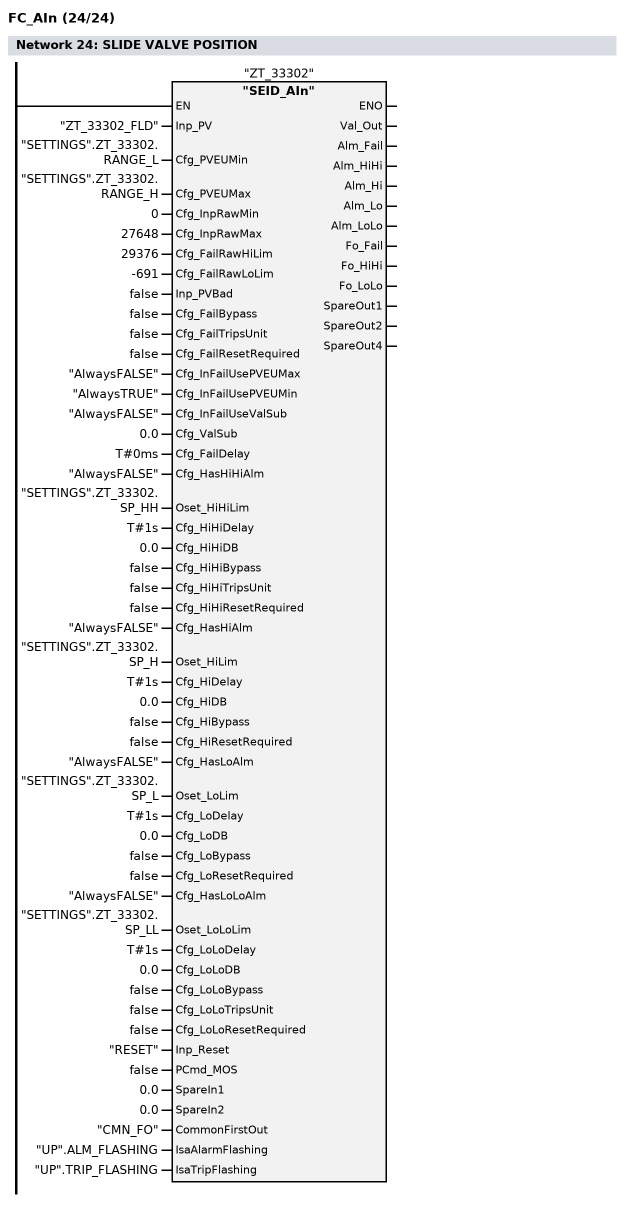
   RUNG wire#powerrail
      "ZT_33302"(Inp_PV := "ZT_33302_FLD", Cfg_PVEUMin := "SETTINGS".ZT_33302.RANGE_L, Cfg_PVEUMax := "SETTINGS".ZT_33302.RANGE_H, Cfg_InpRawMin := 0, Cfg_InpRawMax := 27648, Cfg_FailRawHiLim := 29376, Cfg_FailRawLoLim := -691, Inp_PVBad := false, Cfg_FailBypass := false, Cfg_FailTripsUnit := false, Cfg_FailResetRequired := false, Cfg_InFailUsePVEUMax := "AlwaysFALSE", Cfg_InFailUsePVEUMin := "AlwaysTRUE", Cfg_InFailUseValSub := "AlwaysFALSE", Cfg_ValSub := 0.0, Cfg_FailDelay := T#0ms, Cfg_HasHiHiAlm := "AlwaysFALSE", Oset_HiHiLim := "SETTINGS".ZT_33302.SP_HH, Cfg_HiHiDelay := T#1s, Cfg_HiHiDB := 0.0, Cfg_HiHiBypass := false, Cfg_HiHiTripsUnit := false, Cfg_HiHiResetRequired := false, Cfg_HasHiAlm := "AlwaysFALSE", Oset_HiLim := "SETTINGS".ZT_33302.SP_H, Cfg_HiDelay := T#1s, Cfg_HiDB := 0.0, Cfg_HiBypass := false, Cfg_HiResetRequired := false, Cfg_HasLoAlm := "AlwaysFALSE", Oset_LoLim := "SETTINGS".ZT_33302.SP_L, Cfg_LoDelay := T#1s, Cfg_LoDB := 0.0, Cfg_LoBypass := false, Cfg_LoResetRequired := false, Cfg_HasLoLoAlm := "AlwaysFALSE", Oset_LoLoLim := "SETTINGS".ZT_33302.SP_LL, Cfg_LoLoDelay := T#1s, Cfg_LoLoDB := 0.0, Cfg_LoLoBypass := false, Cfg_LoLoTripsUnit := false, Cfg_LoLoResetRequired := false, Inp_Reset := "RESET", PCmd_MOS := false, SpareIn1 := 0.0, SpareIn2 := 0.0, CommonFirstOut := "CMN_FO", IsaAlarmFlashing := "UP".ALM_FLASHING, IsaTripFlashing := "UP".TRIP_FLASHING, Val_Out =>, Alm_Fail =>, Alm_HiHi =>, Alm_Hi =>, Alm_Lo =>, Alm_LoLo =>, Fo_Fail =>, Fo_HiHi =>, Fo_LoLo =>, SpareOut1 =>, SpareOut2 =>, SpareOut4 =>)
   END_RUNG
   // the same network as SCL:
   "ZT_33302"(Inp_PV := "ZT_33302_FLD",   // "SEID_AIn"
              Cfg_PVEUMin := "SETTINGS".ZT_33302.RANGE_L,
              Cfg_PVEUMax := "SETTINGS".ZT_33302.RANGE_H,
              Cfg_InpRawMin := 0,
              Cfg_InpRawMax := 27648,
              Cfg_FailRawHiLim := 29376,
              Cfg_FailRawLoLim := -691,
              Inp_PVBad := false,
              Cfg_FailBypass := false,
              Cfg_FailTripsUnit := false,
              Cfg_FailResetRequired := false,
              Cfg_InFailUsePVEUMax := "AlwaysFALSE",
              Cfg_InFailUsePVEUMin := "AlwaysTRUE",
              Cfg_InFailUseValSub := "AlwaysFALSE",
              Cfg_ValSub := 0.0,
              Cfg_FailDelay := T#0ms,
              Cfg_HasHiHiAlm := "AlwaysFALSE",
              Oset_HiHiLim := "SETTINGS".ZT_33302.SP_HH,
              Cfg_HiHiDelay := T#1s,
              Cfg_HiHiDB := 0.0,
              Cfg_HiHiBypass := false,
              Cfg_HiHiTripsUnit := false,
              Cfg_HiHiResetRequired := false,
              Cfg_HasHiAlm := "AlwaysFALSE",
              Oset_HiLim := "SETTINGS".ZT_33302.SP_H,
              Cfg_HiDelay := T#1s,
              Cfg_HiDB := 0.0,
              Cfg_HiBypass := false,
              Cfg_HiResetRequired := false,
              Cfg_HasLoAlm := "AlwaysFALSE",
              Oset_LoLim := "SETTINGS".ZT_33302.SP_L,
              Cfg_LoDelay := T#1s,
              Cfg_LoDB := 0.0,
              Cfg_LoBypass := false,
              Cfg_LoResetRequired := false,
              Cfg_HasLoLoAlm := "AlwaysFALSE",
              Oset_LoLoLim := "SETTINGS".ZT_33302.SP_LL,
              Cfg_LoLoDelay := T#1s,
              Cfg_LoLoDB := 0.0,
              Cfg_LoLoBypass := false,
              Cfg_LoLoTripsUnit := false,
              Cfg_LoLoResetRequired := false,
              Inp_Reset := "RESET",
              PCmd_MOS := false,
              SpareIn1 := 0.0,
              SpareIn2 := 0.0,
              CommonFirstOut := "CMN_FO",
              IsaAlarmFlashing := "UP".ALM_FLASHING,
              IsaTripFlashing := "UP".TRIP_FLASHING);
END_REGION
END_FUNCTION
